(* CODESYS project INTERNA2 DRIVE TEST V17.project

Project tree, tasks and I/O mapping:
  Device : TX510-P3CV01, Turck, order no. 6828105, version 1.0.4.0
    application Application
      libraries: Standard, * (System); VisuDialogs, * (System); CAA File, * (CAA Technical Workgroup); CAA Real Time Clock Extern, * (CAA Technical Workgroup); SysTime23, 3.5.2.0 (System); NETWORK, 1.2.1.0 (OSCAT); SysTimeCore, * (System)
      task VISU_TASK (cyclic, interval 100 ms, priority 31) calls VisuElems.Visu_Prg
      task ENIPScannerServiceTask (cyclic, interval t#20ms, priority 30) calls EtherNet_IP_Scanner.ServiceCycle
      task MainTask (cyclic, interval t#20ms, priority 1) calls PLC_PRG
      task ENIPScannerIOTask (cyclic, interval t#10ms, priority 1) calls EtherNet_IP_Scanner.IOCycle
      task AlarmManagerTask (cyclic, interval 50 ms, priority 31) calls AlarmManager.Alarm_Prg
      visualisation PRINCIPAL
      visualisation Analog_Test
      visualisation Drive_Test
      program PLC_PRG [LD]
      global variables GLOBAL_VARS
      visualisation Test_DAQ
      program CSVMON_FILE_GEN [LD]
      Alarm Configuration
        alarm class Error (priority 10, acknowledge ACK)
        alarm class Warning (priority 30, acknowledge REP)
        alarm class Info (priority 100, acknowledge REP)
        AlarmStorage
        text list AlarmGroup
        alarm group AlarmGroup
            11 [Info]: Comparison Equal, ExpressionToCompare TRUE, Expression OPERACION.ROTADORES_INFO_MSG - "PARA ACCIONAR ROTADORES, MUEVA EL BUGGY HACIA EL SUR"
            8 [Info]: Comparison Equal, ExpressionToCompare TRUE, Expression PLC_PRG.ANY_ALARM - "PRESIONE EL BOTON CONFIRMAR PARA RESTABLECER"
            9 [Error]: Comparison Equal, ExpressionToCompare TRUE, Expression PLC_PRG.POWERFLEX_FAULT_ACTIVE - "FALLA DRIVE MOTOR BUGGY "
            19 [Info]: Comparison Equal, ExpressionToCompare TRUE, Expression PLC_PRG.HMI_AUTO_MODE - "INFO MODO AUTO: BUGGY DIRECCION NORTE, VELOCIDAD LENTA"
            10 [Error]: Comparison Equal, ExpressionToCompare TRUE, Expression PLC_PRG.REMOTE_MODULE2_FAULT - "L1: ERROR COMUNICACION MODULO GABINETE VARIADOR & FUERZA"
            15 [Warning]: Comparison Equal, ExpressionToCompare FALSE, Expression OPERACION.SW_ANTORCHA_EJEB - "LIMITE CABEZAL ANTORCHA EJEB ALCANZADO"
            18 [Error]: Comparison Equal, ExpressionToCompare TRUE, Expression PLC_PRG.WELDING_TRAVEL_FEEDBACK_FAULT - "ERROR EN GENERACION DE ARCO"
            16 [Warning]: Comparison Equal, ExpressionToCompare FALSE, Expression OPERACION.SW_BOOM_UP - "LIMITE BOOM SUPERIOR ALCANZADO"
            17 [Warning]: Comparison Equal, ExpressionToCompare FALSE, Expression OPERACION.SW_BOOM_DOWN - "LIMITE BOOM INFERIOR ALCANZADO"
            3 [Error]: Comparison Equal, ExpressionToCompare TRUE, Expression PLC_PRG.ENCODER_FAULT - "ERROR DE SINCRONIZACION BUGGY:REVISAR ENCODER"
            4 [Warning]: Comparison Equal, ExpressionToCompare FALSE, Expression PLC_PRG.SW_NORTE - "BUGGY LIMTE DE CARRERA NORTE ALCANZADO"
            5 [Warning]: Comparison Equal, ExpressionToCompare FALSE, Expression PLC_PRG.SW_SUR - "BUGGY LIMITE DE CARRERA SUR ALCANZADO"
            6 [Error]: Comparison Equal, ExpressionToCompare TRUE, Expression PLC_PRG.REMOTE_MODULE1_FAULT - "L0: ERROR COMUNICACION MODULO DETRAS HMI PRINCIPAL"
            7 [Warning]: Comparison Equal, ExpressionToCompare TRUE, Expression PLC_PRG.EMERGENCY_STOP_ACTIVE - "PARO DE EMERGENCIA EXTERNO ACTIVO"
            14 [Warning]: Comparison Equal, ExpressionToCompare FALSE, Expression OPERACION.SW_ANTORCHA_EJEA - "LIMITE CABEZAL ANTORCHA EJEA ALCANZADO"
            13 [Warning]: Comparison Equal, ExpressionToCompare FALSE, Expression OPERACION.SW_ANTORCHA_DOWN - "LIMITE CABEZAL ANTORCHA INFERIOR ALCANZADO"
            12 [Warning]: Comparison Equal, ExpressionToCompare FALSE, Expression OPERACION.SW_ANORTCHA_UP - "LIMITE CABEZAL ANTORCHA SUPERIOR ALCANZADO"
            20 [Error]: Comparison Equal, ExpressionToCompare TRUE, Expression PLC_PRG.REMOTE_MODULE3_FAULT - "L2: ERROR COMUNICACION MODULO GABINETE AUXILIAR,ANTORCHAS"
      program OPERACION [LD]
      visualisation OPERACION
      visualisation BUGGY
    Ethernet : Ethernet, Turck, version 3.5.7.20
        settings: IPAddress = [192,168,5,211]; SubnetMask = [255,255,255,0]; GatewayAddress = [0,0,0,0]; MACAddress = [16#00,16#00,16#00,16#00,16#00,16#00]; SaveCommunicationSettings = FALSE
      EtherNet_IP_Scanner : EtherNet/IP Scanner, 3S - Smart Software Solutions GmbH, order no. 1, version 3.5.7.0
          settings: IPAddress = [16#C0,16#A8,16#05,16#65]; SubnetMask = [16#00,16#00,16#00,16#00]; GatewayAddress = [16#00,16#00,16#00,16#00]; TCPFlags = 1; Options.Auto-Reestablish Connections = True
        REMOTE_MODULE1 : BL20-E-GW-EN, TURCK, order no. 6827329, version Major Revision=16#2, Minor Revision = 16#7
            settings: INITIALIZED = TRUE; IP address of Target = [16#C0,16#A8,16#05,16#67]; Keying.Compatibility Bit = TRUE; RequiredConfigVersion = 50660864; Number of Connections = 1; Connection Settings.Requested packet intervall (µs) = 10000; Connection Settings.OT Connection Parameters = 18442; Connection Settings.TO Connection Parameters = 10246; Connection Settings.Connection Flags = 1056; Connection Settings.Connection Path Size = 8; Connection Settings.Config#2 Size = 16; Configuration Data = [16#0,16#0,16#0,16#0,16#0,16#0,16#0,16#0,16#0,16#0,16#0,16#0,16#0,16#0,16#0,16#0]; Connection Path = [16#20,16#04,16#24,16#6A,16#2C,16#66,16#2C,16#65]; DI1_0_RESERVED.ReadOnly = False; DI1_0_RESERVED.BitSize = 16; DI1_0_RESERVED.DataSize = 2; DI1_1.ReadOnly = False; DI1_1.BitSize = 16; DI1_1.DataSize = 2; DO1_0_RESERVED.ReadOnly = False; DO1_0_RESERVED.BitSize = 16; DO1_0_RESERVED.DataSize = 2; D01_1.ReadOnly = False; D01_1.BitSize = 16; D01_1.DataSize = 2; DI1_0_RESERVED.Name = 'DI1_0_RESERVED'; DI1_0_RESERVED.HelpString = ''; DI1_0_RESERVED.ReadOnly = False; DI1_0_RESERVED.BitSize = 16; DI1_0_RESERVED.DataSize = 2; DI1_0_RESERVED.DataType = 'UINT'; DI1_1.Name = 'DI1_1'; DI1_1.HelpString = ''; DI1_1.ReadOnly = False; DI1_1.BitSize = 16; DI1_1.DataSize = 2; DI1_1.DataType = 'UINT'; DO1_0_RESERVED.Name = 'DO1_0_RESERVED'; DO1_0_RESERVED.HelpString = ''; DO1_0_RESERVED.ReadOnly = False;
              DO1_0_RESERVED.BitSize = 16; DO1_0_RESERVED.DataSize = 2; DO1_0_RESERVED.DataType = 'UINT'; D01_1.Name = 'D01_1'; D01_1.HelpString = ''; D01_1.ReadOnly = False; D01_1.BitSize = 16; D01_1.DataSize = 2; D01_1.DataType = 'UINT'; ConfigVersion = 50660864
            input  Application.PLC_PRG.EMERGENCY_STOP : BOOL  // DI1_1.Bit0
            input  Application.OPERACION.JOYUP : BOOL  // DI1_1.Bit1
            input  Application.OPERACION.JOYDOWN : BOOL  // DI1_1.Bit2
            input  Application.OPERACION.JOY_EJEA : BOOL  // DI1_1.Bit3
            input  Application.OPERACION.JOY_EJEB : BOOL  // DI1_1.Bit4
            input  Application.PLC_PRG.NA4_TRAVEL2 : BOOL  // DI1_1.Bit12
            input  Application.PLC_PRG.NA4_TRAVEL1 : BOOL  // DI1_1.Bit13
            input  Application.PLC_PRG.NA5_TRAVEL : BOOL  // DI1_1.Bit14
            input  Application.PLC_PRG.HEARTBEAT_RETURN : BOOL  // DI1_1.Bit15
            output Application.PLC_PRG.NA5_START : BOOL  // D01_1.Bit0
            output Application.PLC_PRG.NA4_START1 : BOOL  // D01_1.Bit1
            output Application.PLC_PRG.NA4_START2 : BOOL  // D01_1.Bit2
            output Application.PLC_PRG.NA_NOT_STOP : BOOL  // D01_1.Bit3
            output Application.PLC_PRG.HEARTBEAT_SEND : BOOL  // D01_1.Bit15
            unmapped channels: DI1_0_RESERVED, DI1_1, DO1_0_RESERVED, D01_1
        BUGGY_DRIVE : PowerFlex 525, Rockwell Automation - Allen-Bradley, order no. 25B..., version Major Revision=16#4, Minor Revision = 16#1
            settings: INITIALIZED = TRUE; IP address of Target = [16#C0,16#A8,16#05,16#66]; Keying.Check Vendor Code = FALSE; Keying.Check Product Code = FALSE; RequiredConfigVersion = 50660864; Number of Connections = 1; Connection Settings.Requested packet intervall (µs) = 10000; Connection Settings.OT Connection Parameters = 18442; Connection Settings.TO Connection Parameters = 18442; Connection Settings.Connection Flags = 1056; Connection Settings.Connection Path Size = 8; Connection Path = [16#20,16#04,16#24,16#06,16#2C,16#02,16#2C,16#01]; Reserved.ReadOnly = False; Reserved.BitSize = 32; Reserved.DataSize = 4; Logic Status 0.ReadOnly = False; Logic Status 0.BitSize = 16; Logic Status 0.DataSize = 2; Feedback 0.ReadOnly = False; Feedback 0.BitSize = 16; Feedback 0.DataSize = 2; Logic Command 0.ReadOnly = False; Logic Command 0.BitSize = 16; Logic Command 0.DataSize = 2; Reference 0.ReadOnly = False; Reference 0.BitSize = 16; Reference 0.DataSize = 2; Reserved.Name = 'Reserved'; Reserved.HelpString = ''; Reserved.ReadOnly = False; Reserved.BitSize = 32; Reserved.DataSize = 4; Reserved.DataType = 'DWORD'; Logic Status 0.Name = 'Logic Status 0'; Logic Status 0.HelpString = 'Drive 0 Logic Status'; Logic Status 0.ReadOnly = False; Logic Status 0.BitSize = 16; Logic Status 0.DataSize = 2; Logic Status 0.DataType = 'WORD'; Feedback 0.Name = 'Feedback 0';
              Feedback 0.HelpString = 'Drive 0 Feedback'; Feedback 0.ReadOnly = False; Feedback 0.BitSize = 16; Feedback 0.DataSize = 2; Feedback 0.DataType = 'WORD'; Logic Command 0.Name = 'Logic Command 0'; Logic Command 0.HelpString = 'Drive 0 Logic Command'; Logic Command 0.ReadOnly = False; Logic Command 0.BitSize = 16; Logic Command 0.DataSize = 2; Logic Command 0.DataType = 'WORD'; Reference 0.Name = 'Reference 0'; Reference 0.HelpString = 'Drive 0 Reference'; Reference 0.ReadOnly = False; Reference 0.BitSize = 16; Reference 0.DataSize = 2; Reference 0.DataType = 'WORD'; ConfigVersion = 50660864
            input  Application.PLC_PRG.PWRFLEX_LOGIC_STATUS : WORD  // Logic Status 0
            input  Application.PLC_PRG.PWRFLEX_FEEDBACK : WORD  // Feedback 0
            output Application.PLC_PRG.PWRFLEX_LOGIC_CMD : WORD  // Logic Command 0
            output Application.PLC_PRG.PWRFLEX_SPEEDREF : WORD  // Reference 0
            unmapped channels: Reserved
        In_Sight_Micro_1000_Series : In-Sight Micro 1000 Series, Cognex, order no. ism1XXX, version Major Revision=16#a, Minor Revision = 16#1
            settings: INITIALIZED = TRUE; IP address of Target = [16#C0,16#A8,16#05,16#04]; Keying.Compatibility Bit = TRUE; RequiredConfigVersion = 50660864; Number of Connections = 1; Connection Settings.Requested packet intervall (µs) = 10000; Connection Settings.OT Connection Parameters = 18434; Connection Settings.TO Connection Parameters = 10258; Connection Settings.Connection Flags = 1062; Connection Settings.Connection Path Size = 8; Connection Path = [16#20,16#04,16#24,16#01,16#2C,16#FE,16#2C,16#0C]; Generic Parameter1.ReadOnly = False; Generic Parameter1.BitSize = 32; Generic Parameter1.DataSize = 4; Generic Parameter3.ReadOnly = False; Generic Parameter3.BitSize = 32; Generic Parameter3.DataSize = 4; Generic Parameter2.ReadOnly = False; Generic Parameter2.BitSize = 32; Generic Parameter2.DataSize = 4; Generic Parameter4.ReadOnly = False; Generic Parameter4.BitSize = 32; Generic Parameter4.DataSize = 4; Generic Parameter1.Name = 'Generic Parameter1'; Generic Parameter1.HelpString = ''; Generic Parameter1.ReadOnly = False; Generic Parameter1.BitSize = 32; Generic Parameter1.DataSize = 4; Generic Parameter1.DataType = 'REAL'; Generic Parameter3.Name = 'Generic Parameter3'; Generic Parameter3.HelpString = ''; Generic Parameter3.ReadOnly = False; Generic Parameter3.BitSize = 32; Generic Parameter3.DataSize = 4; Generic Parameter3.DataType = 'REAL'; Generic Parameter2.Name = 'Generic Parameter2'; Generic Parameter2.HelpString = ''; Generic Parameter2.ReadOnly = False; Generic Parameter2.BitSize = 32; Generic Parameter2.DataSize = 4;
              Generic Parameter2.DataType = 'REAL'; Generic Parameter4.Name = 'Generic Parameter4'; Generic Parameter4.HelpString = ''; Generic Parameter4.ReadOnly = False; Generic Parameter4.BitSize = 32; Generic Parameter4.DataSize = 4; Generic Parameter4.DataType = 'REAL'; ConfigVersion = 50660864
            input  Application.PLC_PRG.COGNEX_AUX1 : REAL  // Generic Parameter1
            input  Application.PLC_PRG.COGNEX_AUX2 : REAL  // Generic Parameter3
            input  Application.PLC_PRG.COGNEX_AUX3 : REAL  // Generic Parameter2
            input  Application.PLC_PRG.COGNEX_AUX4 : REAL  // Generic Parameter4
        REMOTE_MODULE2 : BL20-E-GW-EN, TURCK, order no. 6827329, version Major Revision=16#2, Minor Revision = 16#7
            settings: INITIALIZED = TRUE; IP address of Target = [16#C0,16#A8,16#05,16#69]; Keying.Compatibility Bit = TRUE; RequiredConfigVersion = 50660864; Number of Connections = 1; Connection Settings.Requested packet intervall (µs) = 10000; Connection Settings.OT Connection Parameters = 18442; Connection Settings.TO Connection Parameters = 10246; Connection Settings.Connection Flags = 1056; Connection Settings.Connection Path Size = 8; Connection Settings.Config#2 Size = 16; Configuration Data = [16#0,16#0,16#0,16#0,16#0,16#0,16#0,16#0,16#0,16#0,16#0,16#0,16#0,16#0,16#0,16#0]; Connection Path = [16#20,16#04,16#24,16#6A,16#2C,16#66,16#2C,16#65]; DI2_0_RESERVED.ReadOnly = False; DI2_0_RESERVED.BitSize = 16; DI2_0_RESERVED.DataSize = 2; DI2_1.ReadOnly = False; DI2_1.BitSize = 16; DI2_1.DataSize = 2; DO2_0_RESERVED.ReadOnly = False; DO2_0_RESERVED.BitSize = 16; DO2_0_RESERVED.DataSize = 2; DO2_1.ReadOnly = False; DO2_1.BitSize = 16; DO2_1.DataSize = 2; DI2_0_RESERVED.Name = 'DI2_0_RESERVED'; DI2_0_RESERVED.HelpString = ''; DI2_0_RESERVED.ReadOnly = False; DI2_0_RESERVED.BitSize = 16; DI2_0_RESERVED.DataSize = 2; DI2_0_RESERVED.DataType = 'UINT'; DI2_1.Name = 'DI2_1'; DI2_1.HelpString = ''; DI2_1.ReadOnly = False; DI2_1.BitSize = 16; DI2_1.DataSize = 2; DI2_1.DataType = 'UINT'; DO2_0_RESERVED.Name = 'DO2_0_RESERVED'; DO2_0_RESERVED.HelpString = ''; DO2_0_RESERVED.ReadOnly = False;
              DO2_0_RESERVED.BitSize = 16; DO2_0_RESERVED.DataSize = 2; DO2_0_RESERVED.DataType = 'UINT'; DO2_1.Name = 'DO2_1'; DO2_1.HelpString = ''; DO2_1.ReadOnly = False; DO2_1.BitSize = 16; DO2_1.DataSize = 2; DO2_1.DataType = 'UINT'; ConfigVersion = 50660864
            input  Application.OPERACION.SW_BOOM_DOWN : BOOL  // DI2_1.Bit0
            input  Application.OPERACION.SW_BOOM_UP : BOOL  // DI2_1.Bit1
            input  Application.PLC_PRG.HEARTBEAT_RETURN2 : BOOL  // DI2_1.Bit15
            output Application.OPERACION.CONVEYOR_NORTE_L02_KM1 : BOOL  // DO2_1.Bit0
            output Application.OPERACION.CONVEYOR_SUR_L02_KM2 : BOOL  // DO2_1.Bit1
            output Application.OPERACION.ROTADORES_EJEA_L02_KM3 : BOOL  // DO2_1.Bit2
            output Application.OPERACION.ROTADORES_EJEB_L02_KM4 : BOOL  // DO2_1.Bit3
            output Application.OPERACION.BOOM_DOWN_KM6 : BOOL  // DO2_1.Bit4
            output Application.OPERACION.BOOM_UP_KM5 : BOOL  // DO2_1.Bit5
            output Application.OPERACION.ASPIRADORA_KM7 : BOOL  // DO2_1.Bit6
            output Application.OPERACION.RELAY_BRAZO_TIERRAS_UP : BOOL  // DO2_1.Bit7
            output Application.OPERACION.RELAY_BRAZO_TIERRAS_DOWN : BOOL  // DO2_1.Bit8
            output Application.PLC_PRG.HEARTBEAT_SEND2 : BOOL  // DO2_1.Bit15
            unmapped channels: DI2_0_RESERVED, DI2_1, DO2_0_RESERVED, DO2_1
        REMOTE_MODULE3 : BL20-E-GW-EN, TURCK, order no. 6827329, version Major Revision=16#2, Minor Revision = 16#7
            settings: INITIALIZED = TRUE; IP address of Target = [16#C0,16#A8,16#05,16#6A]; Keying.Compatibility Bit = TRUE; RequiredConfigVersion = 50660864; Number of Connections = 1; Connection Settings.Requested packet intervall (µs) = 10000; Connection Settings.OT Connection Parameters = 18442; Connection Settings.TO Connection Parameters = 18438; Connection Settings.Connection Flags = 1056; Connection Settings.Connection Path Size = 8; Connection Settings.Config#2 Size = 16; Configuration Data = [16#0,16#0,16#0,16#0,16#0,16#0,16#0,16#0,16#0,16#0,16#0,16#0,16#0,16#0,16#0,16#0]; Connection Path = [16#20,16#04,16#24,16#6A,16#2C,16#66,16#2C,16#65]; DI3_0_RESERVED.ReadOnly = False; DI3_0_RESERVED.BitSize = 16; DI3_0_RESERVED.DataSize = 2; DI3_1.ReadOnly = False; DI3_1.BitSize = 16; DI3_1.DataSize = 2; DO3_0_RESERVED.ReadOnly = False; DO3_0_RESERVED.BitSize = 16; DO3_0_RESERVED.DataSize = 2; DO3_1.ReadOnly = False; DO3_1.BitSize = 16; DO3_1.DataSize = 2; DI3_0_RESERVED.Name = 'DI3_0_RESERVED'; DI3_0_RESERVED.HelpString = ''; DI3_0_RESERVED.ReadOnly = False; DI3_0_RESERVED.BitSize = 16; DI3_0_RESERVED.DataSize = 2; DI3_0_RESERVED.DataType = 'UINT'; DI3_1.Name = 'DI3_1'; DI3_1.HelpString = ''; DI3_1.ReadOnly = False; DI3_1.BitSize = 16; DI3_1.DataSize = 2; DI3_1.DataType = 'UINT'; DO3_0_RESERVED.Name = 'DO3_0_RESERVED'; DO3_0_RESERVED.HelpString = ''; DO3_0_RESERVED.ReadOnly = False;
              DO3_0_RESERVED.BitSize = 16; DO3_0_RESERVED.DataSize = 2; DO3_0_RESERVED.DataType = 'UINT'; DO3_1.Name = 'DO3_1'; DO3_1.HelpString = ''; DO3_1.ReadOnly = False; DO3_1.BitSize = 16; DO3_1.DataSize = 2; DO3_1.DataType = 'UINT'; ConfigVersion = 50660864
            input  Application.PLC_PRG.SW_NORTE : BOOL  // DI3_1.Bit0
            input  Application.PLC_PRG.SW_SUR : BOOL  // DI3_1.Bit1
            input  Application.OPERACION.SW_ANORTCHA_UP : BOOL  // DI3_1.Bit2
            input  Application.OPERACION.SW_ANTORCHA_DOWN : BOOL  // DI3_1.Bit3
            input  Application.OPERACION.SW_ANTORCHA_EJEA : BOOL  // DI3_1.Bit4
            input  Application.OPERACION.SW_ANTORCHA_EJEB : BOOL  // DI3_1.Bit5
            input  Application.PLC_PRG.HEARTBEAT_RETURN3 : BOOL  // DI3_1.Bit15
            output Application.OPERACION.RELAY_VALVULA1 : BOOL  // DO3_1.Bit0
            output Application.OPERACION.RELAY_VALVULA2 : BOOL  // DO3_1.Bit1
            output Application.OPERACION.TOLVA_ON : BOOL  // DO3_1.Bit4
            output Application.OPERACION.CAMARA_ON : BOOL  // DO3_1.Bit5
            output Application.OPERACION.ANTORCHA_EJEA : BOOL  // DO3_1.Bit6
            output Application.OPERACION.ANTORCHA_EJEB : BOOL  // DO3_1.Bit7
            output Application.OPERACION.ANTORCHA_UP : BOOL  // DO3_1.Bit8
            output Application.OPERACION.ANTORCHA_DOWN : BOOL  // DO3_1.Bit9
            output Application.PLC_PRG.HEARTBEAT_SEND3 : BOOL  // DO3_1.Bit15
            unmapped channels: DI3_0_RESERVED, DI3_1, DO3_0_RESERVED, DO3_1
  libraries: VisuSymbols, 3.5.10.0 (System)
  text list GlobalTextList
  text list System
*)

// Device/Application/GLOBAL_VARS
{attribute 'qualified_only'}
VAR_GLOBAL
	  uiFileStdState:     UINT;  //TEXT CMD STATE
	  sFileName: 		  STRING;		//FILE NAM STRING (DIRECTORY+DATA)
	  sFileWriteString:	  STRING;
	
	  
END_VAR

// Device/Application/PLC_PRG
PROGRAM PLC_PRG
VAR
(* 
======>instalar librerias:
1)network(OSCAT 1.2.1.0)
2)CAA FILE 3.5.7.0
3) SYSTIME32 3.5.2.0
*)	

//--BL20 VARS--

//EL SIGUIENTE DIRECCIONAMIENTO NO ES RECOMENDADO, LA DIRECCION PUEDE SER REASIGNADA 
//AL AGREGAR UN DISPOSITIVO:
//	IN00 AT %IB102 :BYTE;
//	IN01 AT %IB103 :BYTE;
//-----DIGITAL-----
//INPUTS
DI1_1 :USINT;
//OUTPUTS
DO1_1 :USINT;

//----ANALOG------
//INPUTS
ANA_INPUT1_1 :INT;
ANA_INPUT1_2 :INT;
//OUTPUTS

//VARS
ANA_IN_AUX1 :REAL;
ANA_AMPS :REAL;

ANA_IN_AUX2 :REAL;


//-----------------------------------POWERFLEX VARS-----------------------------------------//
//MISCELLANEUS
PWRFLEX_START_CMD  :UINT; //16bit integer
PWRFLEX_STOP_CMD  :UINT; 
PWRFLEX_SPEEDREF_AUX :REAL;
PWRFLEX_SPEEDREF_AUX2 :REAL;
PWRFLEX_FEEDBACK :UINT;
PWRFLEX_FEEDBACK_AUX :REAL;
PWRFLEX_FEEDBACK_AUX2 :REAL;
PWRFLEX_FEEDBACK_AUX_OFFSET :REAL;

PWRFLEX_FEEDBACK_AUX3 :REAL;
PWRFLEX_FEEDBACK_AUX4 :REAL;

PWRFLEX_AMPS :REAL;
PWRFLEX_giro :BOOL;

PWRFLEX_AMPS_AUX :REAL;

//START =>26
//STOP =>9

//INPUTS
PWRFLEX_LOGIC_STATUS :WORD;

//OUTPUTS
PWRFLEX_LOGIC_CMD :WORD;
PWRFLEX_OPERATOR_START: BOOL;
PWRFLEX_OPERATOR_STOP: BOOL;
HMI_PWRFLEX_OPERATOR_STOP: BOOL;
PWRFLEX_START_STOP :BOOL;
PWRFLEX_SPEEDREF :WORD;

//----------------------------PROGRAM GENERAL MISCELLANEUS VARS------------------------------//
//->SQUARE GEN - PERIOD:1SEG
TIMER1_A: TON;
TIMER1_B: TON;


ALWAYS_OFF :BOOL:=FALSE;
VAR1 :BOOL;
VAR2 :BOOL;
VAR3 :BOOL;
//declare and assign value example
 //VARx :BOOL :=TRUE;

//----------------------------COGNEX VARS------------------------------//
In_Sight_Micro_1000_Series :DWORD;
COGNEX_AUX :DWORD;
COGNEX_AUX1 :REAL;
COGNEX_AUX2 :REAL;
COGNEX_AUX3 :REAL;
COGNEX_AUX4 :REAL;



//----------------------------TEXT VARS------------------------------//
TXT_CMD_ENABLE: BOOL;
TXT_CMD_SELECT: USINT;


TEST_TEXT: STRING;

TEXT: STRING;
TEST_BIT: BOOL;
TEST_BIT2: BOOL;



TON1: TON;
SAMPLING_TRIGGER: BOOL;


//----------------------------ALARMS------------------------------//
(*
ALARM_ERROR1: BOOL;
ALARM_WARNING1: BOOL;
ALARM_INFO1: BOOL;
*)
ACK_ALARM: BOOL;
ANY_ALARM: BOOL:=FALSE;
(*
ALARM_ERROR1_ACTIVE: BOOL;
ALARM_WARNING1_ACTIVE: BOOL;
ALARM_INFO1_ACTIVE: BOOL;
*)
//-----EMERGENCY STOP----
EMERGENCY_STOP: BOOL;
EMERGENCY_STOP_ACTIVE: BOOL;
HMI_EMERGENCY_STOP: BOOL;
HMI_EMERGENCY_STOP_ACTIVE: BOOL;

//----DRIVE FAULT-------
POWERFLEX_FAULT_ACTIVE: BOOL;

//------ENCODER---------
ENCODER_FAULT_TON: TON;
ENCODER_FAULT: BOOL;
ENCODER_FAULT_AUX: BOOL;
PWRFLEX_SPEED_DEVIATION: REAL;

//------LIMIT SWITCH BUGGY
SW_NORTE: BOOL;
SW_NORTE_FAULT: BOOL;
SW_NORTE_FALLING_TRIGGER: F_TRIG;
SW_SUR: BOOL;
SW_SUR_FAULT: BOOL;
SW_SUR_FALLING_TRIGGER: F_TRIG;

BUGGY_NORTE_ENABLE: BOOL;
BUGGY_NORTE_DISABLE: BOOL;
BUGGY_SUR_ENABLE: BOOL;
BUGGY_SUR_DISABLE: BOOL;
BUGGY_SUR_NORTE_ENABLE: BOOL;
BUGGY_SUR_NORTE_DISABLE: BOOL;

//----------REMOTE MODULE COMMUNICATION ERROR------------
//>>MODULE1 (L0)

HEARTBEAT_SEND: BOOL;
HEARTBEAT_RETURN: BOOL;
REMOTE_MODULE1_FAULT: BOOL;
REMOTE_MODULE1_FAULT_AUX: BOOL;

TIMER_HEARTBEAT_FEEDBACK1: TON;
TIMER_HEARTBEAT_FEEDBACK2: TON;

//-----MODULE 2 COMUNICATION ERROR (L1)
HEARTBEAT_SEND2: BOOL;
HEARTBEAT_RETURN2: BOOL;
REMOTE_MODULE2_FAULT: BOOL;
REMOTE_MODULE2_FAULT_AUX: BOOL;

TIMER_HEARTBEAT_FEEDBACK1_2: TON;
TIMER_HEARTBEAT_FEEDBACK2_2: TON;

//-----MODULE 3 COMUNICATION ERROR (L2)
HEARTBEAT_SEND3: BOOL;
HEARTBEAT_RETURN3: BOOL;
REMOTE_MODULE3_FAULT: BOOL;
REMOTE_MODULE3_FAULT_AUX: BOOL;

TIMER_HEARTBEAT_FEEDBACK1_3: TON;
TIMER_HEARTBEAT_FEEDBACK2_3: TON;

//-------WELDING SEQUENCE ERROR
WELDING_TRAVEL_FEEDBACK: TON;
WELDING_TRAVEL_FEEDBACK_FAULT: BOOL;



//-----------------------------
OPERATOR_CONFIRM_ERROR: BOOL;

//-----------------OPERATOR------------------

BUGGY_SPEED_SELECTOR: BOOL;
BUGGY_SPEED_FAST: REAL:=400.0;
BUGGY_SPEED_SLOW: REAL:=30.0;
BUGGY_SPEED: REAL;
BUGGY_SPEED_AUX1: REAL;
BUGGY_SPEED_FEEDBACK_OFFSET: REAL:=1.0;
BUGGY_SPEED_FEEDBACK_OFFSET_AUX: REAL;
BUGGY_SPEED_REFERENCE_OFFSET: REAL:=1.0;
BUGGY_SPEED_REFERENCE_OFFSET_AUX: REAL;

//------------NA CONTROL-------------
HMI_AUTO_MODE: BOOL;
NA_AUTO_MODE: BOOL;

//NA INPUTS
NA5_TRAVEL: BOOL;  //DC WELDING ACTIVE
NA4_TRAVEL1: BOOL; //AC1 WELDING ACTIVE
NA4_TRAVEL2: BOOL; //AC2 WELDING ACTIVE

//OUTPUTS TO NA
NA5_START: BOOL; //DC START
NA4_START1: BOOL; //AC1 START
NA4_START2: BOOL; //AC2 START

ACTIVATE_NA_WELDING_SEQUENCE: BOOL;
ACTIVATE_NA5_DC: TON; //START DELAY DC
ACTIVATE_NA4_AC1: TON; //START DELAY AC1
ACTIVATE_NA4_AC2: TON; //START DELAY AC1

ALL_NA_TRAVEL_OK: BOOL;

NA_NOT_STOP: BOOL; //PLC STOP TO ALL NA´S

//WELDING AUTO MODE
AUTO_MODE_PERMISSIVES_OK: BOOL;
ASPIRADORA_AUTO_ON: BOOL;

AUTO_MODE_ARC_SELECT: BOOL; //FALSE=2 ARCOS, TRUE=3 ARCOS
AUTO_MODE_BYPASS: BOOL; //BYPASS PARA ACTIVAR ARCOS EN MODO MANUAL

END_VAR
VAR // added by the converter: edge detectors and wires of the graphical bodies
    _w1, _w2, _w3, _w4 : BOOL;
END_VAR

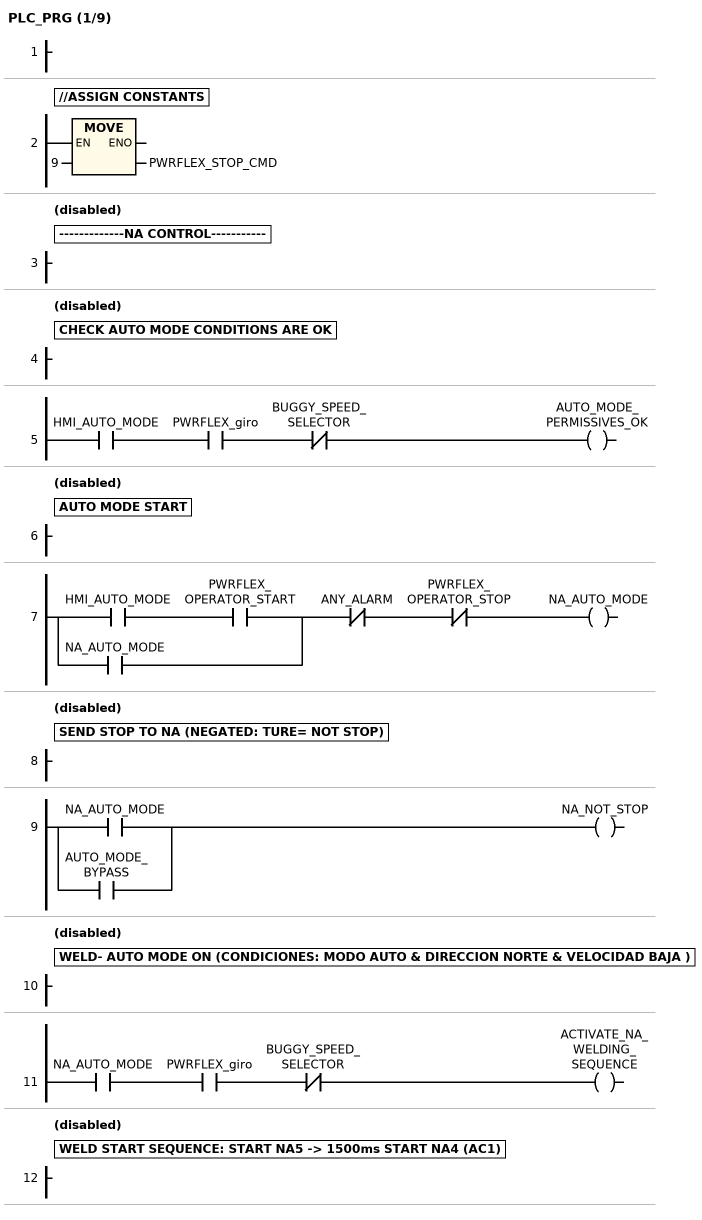
// NETWORK 1

// NETWORK 2
// label: //ASSIGN CONSTANTS
PWRFLEX_STOP_CMD := 9;

// NETWORK 3 (disabled)
// label: -------------NA CONTROL-----------

// NETWORK 4 (disabled)
// label: CHECK AUTO MODE CONDITIONS ARE OK

// NETWORK 5
AUTO_MODE_PERMISSIVES_OK := HMI_AUTO_MODE AND PWRFLEX_giro AND NOT BUGGY_SPEED_SELECTOR;

// NETWORK 6 (disabled)
// label: AUTO MODE START

// NETWORK 7
NA_AUTO_MODE := (HMI_AUTO_MODE AND PWRFLEX_OPERATOR_START OR NA_AUTO_MODE) AND NOT ANY_ALARM AND NOT PWRFLEX_OPERATOR_STOP;

// NETWORK 8 (disabled)
// label: SEND STOP TO NA (NEGATED: TURE= NOT STOP)

// NETWORK 9
NA_NOT_STOP := NA_AUTO_MODE OR AUTO_MODE_BYPASS;

// NETWORK 10 (disabled)
// label: WELD- AUTO MODE ON (CONDICIONES: MODO AUTO & DIRECCION NORTE & VELOCIDAD BAJA )

// NETWORK 11
ACTIVATE_NA_WELDING_SEQUENCE := NA_AUTO_MODE AND PWRFLEX_giro AND NOT BUGGY_SPEED_SELECTOR;

// NETWORK 12 (disabled)
// label: WELD START SEQUENCE: START NA5 -> 1500ms START NA4 (AC1)

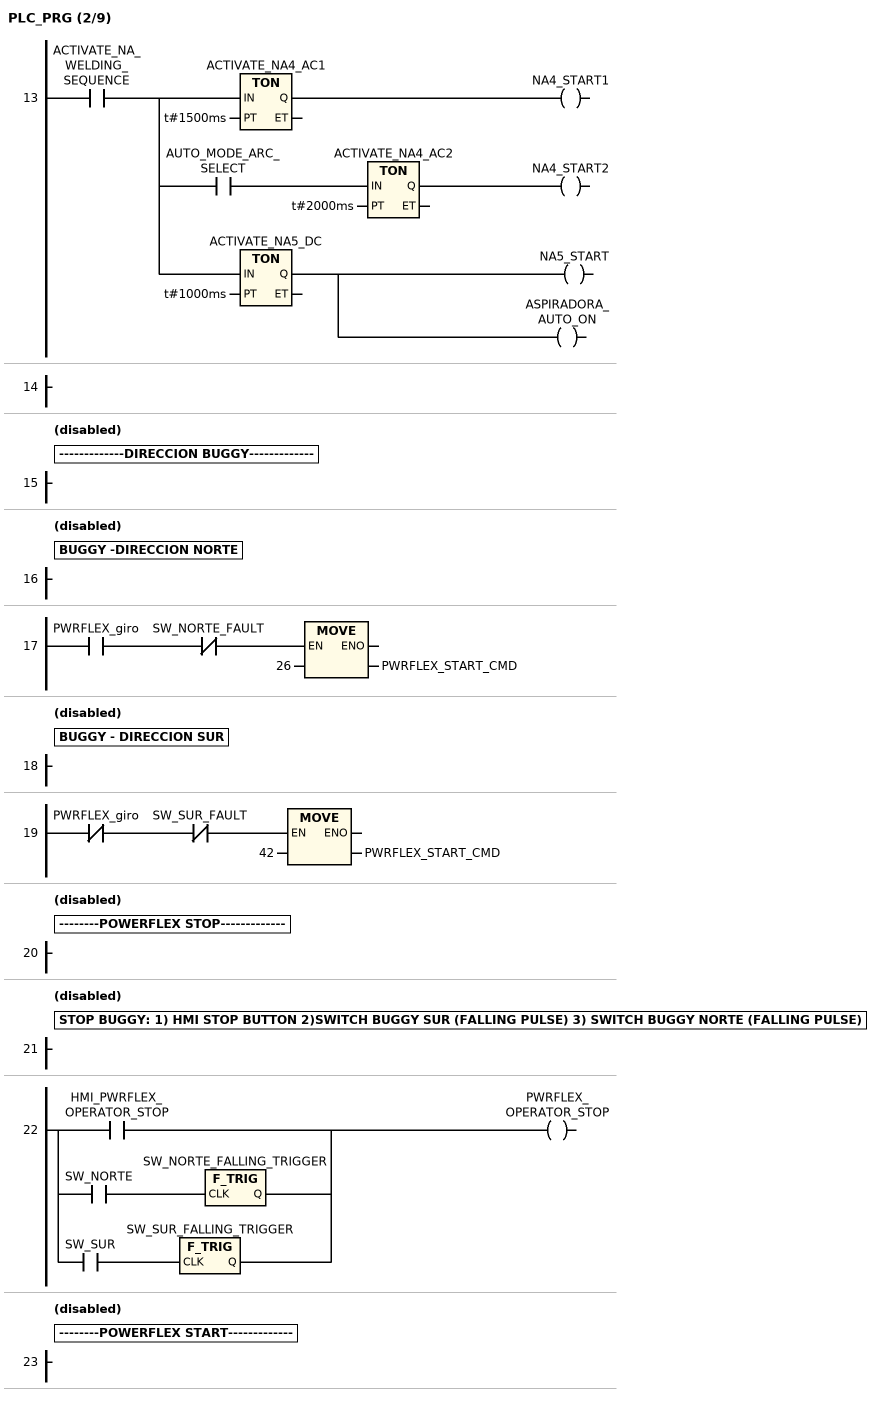
// NETWORK 13
ACTIVATE_NA4_AC1(IN := ACTIVATE_NA_WELDING_SEQUENCE, PT := t#1500ms); // TON
NA4_START1 := ACTIVATE_NA4_AC1.Q;
ACTIVATE_NA4_AC2(IN := ACTIVATE_NA_WELDING_SEQUENCE AND AUTO_MODE_ARC_SELECT, PT := t#2000ms); // TON
NA4_START2 := ACTIVATE_NA4_AC2.Q;
ACTIVATE_NA5_DC(IN := ACTIVATE_NA_WELDING_SEQUENCE, PT := t#1000ms); // TON
NA5_START := ACTIVATE_NA5_DC.Q;
ASPIRADORA_AUTO_ON := ACTIVATE_NA5_DC.Q;

// NETWORK 14

// NETWORK 15 (disabled)
// label: -------------DIRECCION BUGGY-------------

// NETWORK 16 (disabled)
// label: BUGGY -DIRECCION NORTE

// NETWORK 17
IF PWRFLEX_giro AND NOT SW_NORTE_FAULT THEN PWRFLEX_START_CMD := 26; END_IF

// NETWORK 18 (disabled)
// label: BUGGY - DIRECCION SUR

// NETWORK 19
IF NOT PWRFLEX_giro AND NOT SW_SUR_FAULT THEN PWRFLEX_START_CMD := 42; END_IF

// NETWORK 20 (disabled)
// label: --------POWERFLEX STOP-------------

// NETWORK 21 (disabled)
// label: STOP BUGGY: 1) HMI STOP BUTTON 2)SWITCH BUGGY SUR (FALLING PULSE) 3) SWITCH BUGGY NORTE (FALLING PULSE)

// NETWORK 22
SW_NORTE_FALLING_TRIGGER(CLK := SW_NORTE); // F_TRIG
SW_SUR_FALLING_TRIGGER(CLK := SW_SUR); // F_TRIG
PWRFLEX_OPERATOR_STOP := HMI_PWRFLEX_OPERATOR_STOP OR SW_NORTE_FALLING_TRIGGER.Q OR SW_SUR_FALLING_TRIGGER.Q;

// NETWORK 23 (disabled)
// label: --------POWERFLEX START-------------

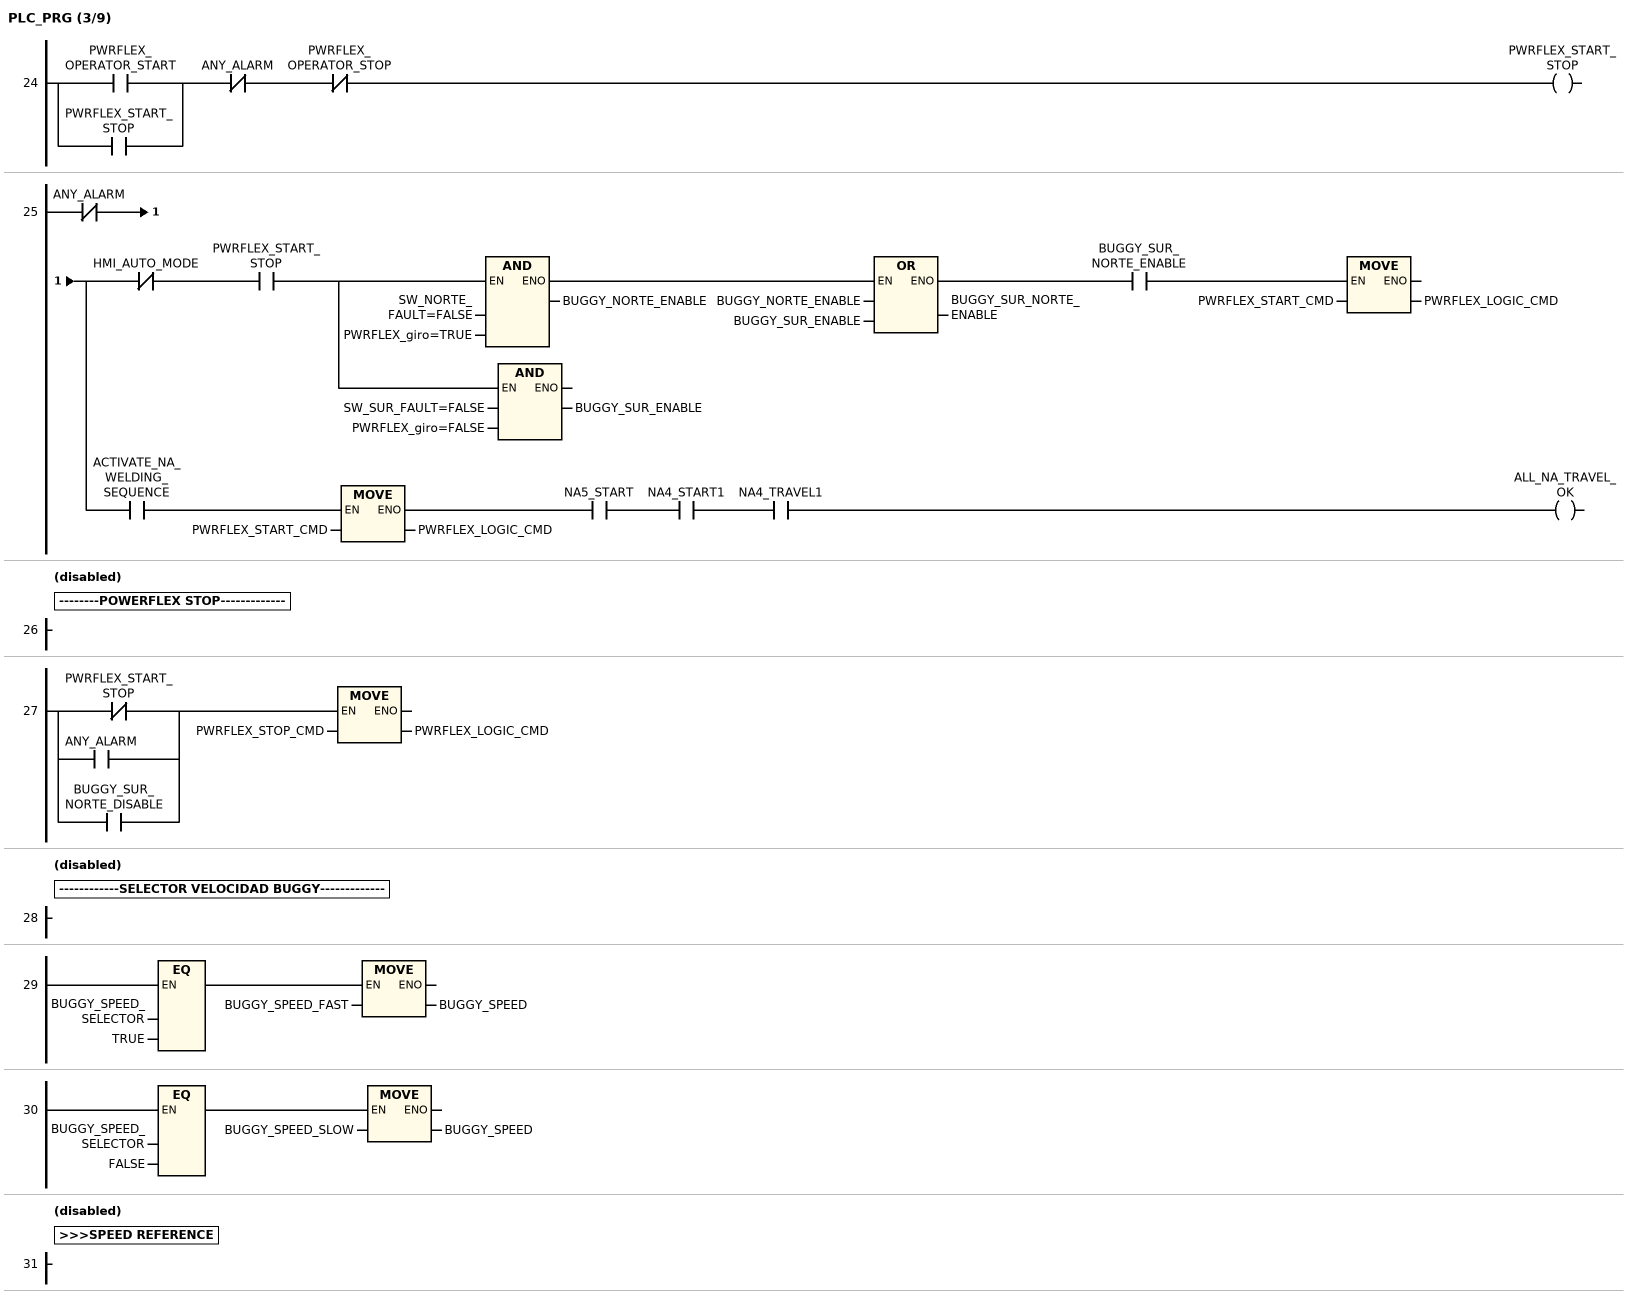
// NETWORK 24
PWRFLEX_START_STOP := (PWRFLEX_OPERATOR_START OR PWRFLEX_START_STOP) AND NOT ANY_ALARM AND NOT PWRFLEX_OPERATOR_STOP;

// NETWORK 25
_w1 := NOT ANY_ALARM;
_w2 := _w1 AND NOT HMI_AUTO_MODE AND PWRFLEX_START_STOP;
IF _w2 THEN BUGGY_NORTE_ENABLE := (SW_NORTE_FAULT=FALSE) AND (PWRFLEX_giro=TRUE); END_IF
IF _w2 THEN BUGGY_SUR_NORTE_ENABLE := BUGGY_NORTE_ENABLE OR BUGGY_SUR_ENABLE; END_IF
IF _w2 AND BUGGY_SUR_NORTE_ENABLE THEN PWRFLEX_LOGIC_CMD := PWRFLEX_START_CMD; END_IF
IF _w2 THEN BUGGY_SUR_ENABLE := (SW_SUR_FAULT=FALSE) AND (PWRFLEX_giro=FALSE); END_IF
IF _w1 AND ACTIVATE_NA_WELDING_SEQUENCE THEN PWRFLEX_LOGIC_CMD := PWRFLEX_START_CMD; END_IF
ALL_NA_TRAVEL_OK := (_w1 AND ACTIVATE_NA_WELDING_SEQUENCE) AND NA5_START AND NA4_START1 AND NA4_TRAVEL1;

// NETWORK 26 (disabled)
// label: --------POWERFLEX STOP-------------

// NETWORK 27
IF NOT PWRFLEX_START_STOP OR ANY_ALARM OR BUGGY_SUR_NORTE_DISABLE THEN
    PWRFLEX_LOGIC_CMD := PWRFLEX_STOP_CMD;
END_IF

// NETWORK 28 (disabled)
// label: ------------SELECTOR VELOCIDAD BUGGY-------------

// NETWORK 29
IF BUGGY_SPEED_SELECTOR = TRUE THEN BUGGY_SPEED := BUGGY_SPEED_FAST; END_IF

// NETWORK 30
IF BUGGY_SPEED_SELECTOR = FALSE THEN BUGGY_SPEED := BUGGY_SPEED_SLOW; END_IF

// NETWORK 31 (disabled)
// label: >>>SPEED REFERENCE

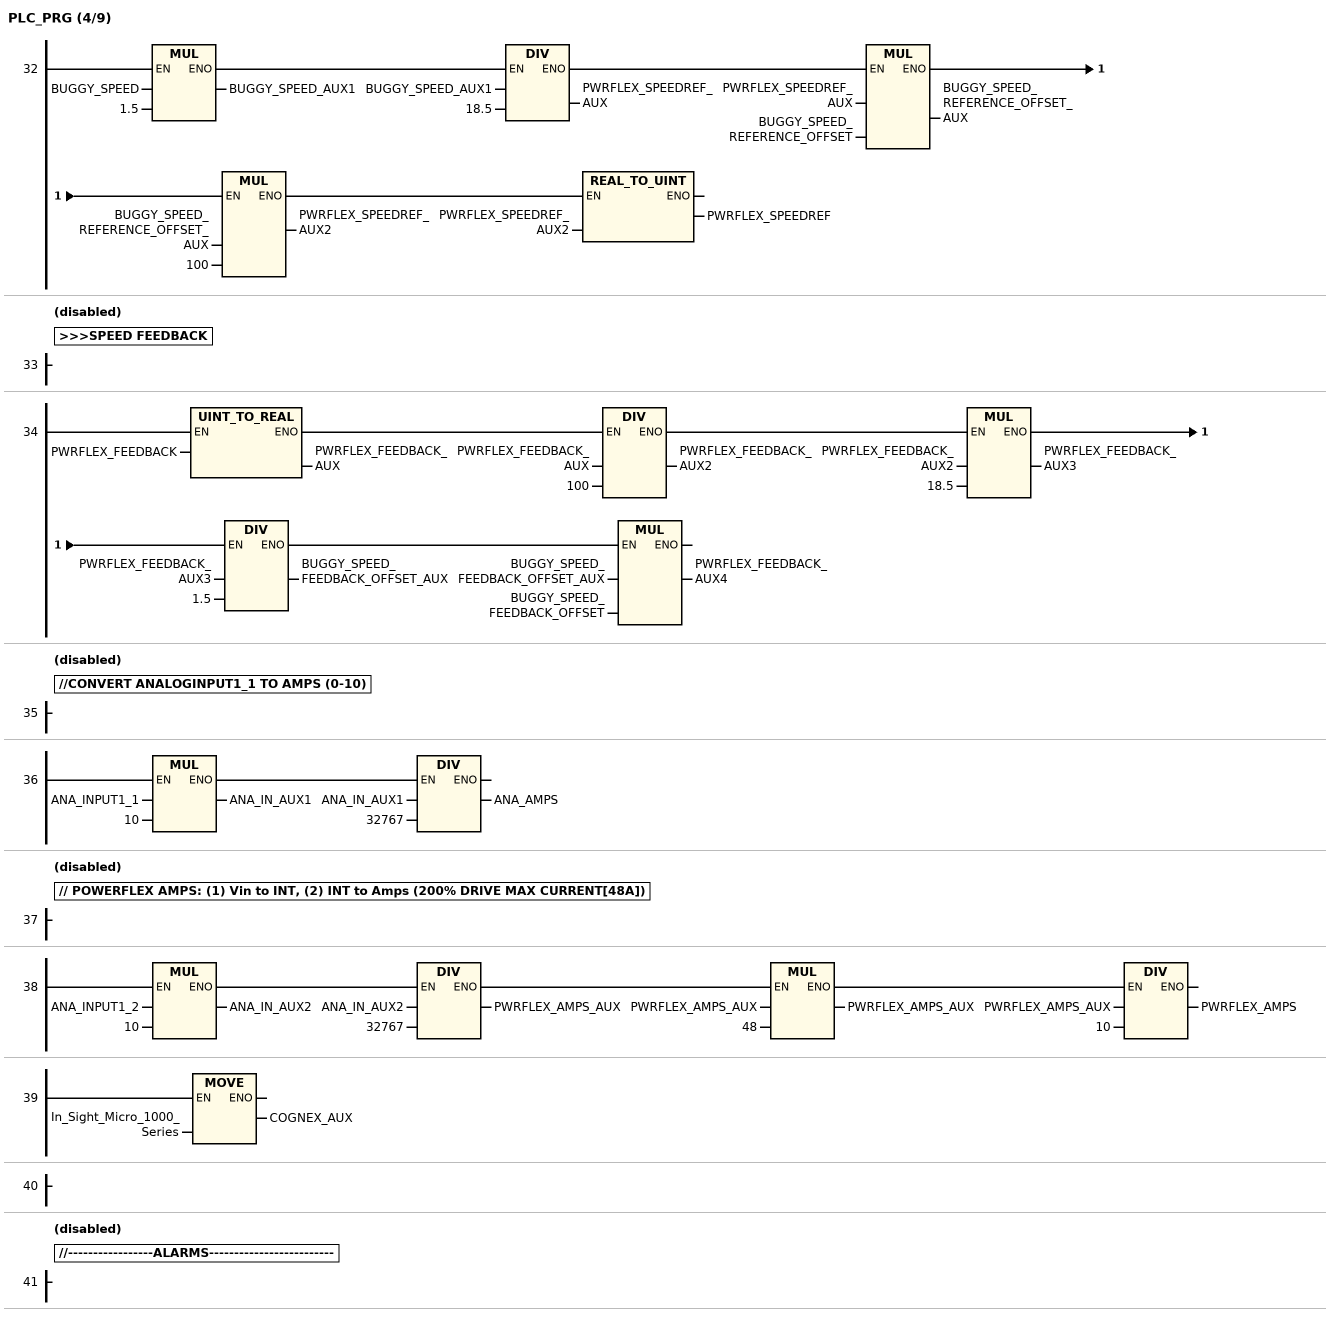
// NETWORK 32
BUGGY_SPEED_AUX1 := BUGGY_SPEED * 1.5;
PWRFLEX_SPEEDREF_AUX := BUGGY_SPEED_AUX1 / 18.5;
BUGGY_SPEED_REFERENCE_OFFSET_AUX := PWRFLEX_SPEEDREF_AUX * BUGGY_SPEED_REFERENCE_OFFSET;
PWRFLEX_SPEEDREF_AUX2 := BUGGY_SPEED_REFERENCE_OFFSET_AUX * 100;
PWRFLEX_SPEEDREF := REAL_TO_UINT(PWRFLEX_SPEEDREF_AUX2);

// NETWORK 33 (disabled)
// label: >>>SPEED FEEDBACK

// NETWORK 34
PWRFLEX_FEEDBACK_AUX := UINT_TO_REAL(PWRFLEX_FEEDBACK);
PWRFLEX_FEEDBACK_AUX2 := PWRFLEX_FEEDBACK_AUX / 100;
PWRFLEX_FEEDBACK_AUX3 := PWRFLEX_FEEDBACK_AUX2 * 18.5;
BUGGY_SPEED_FEEDBACK_OFFSET_AUX := PWRFLEX_FEEDBACK_AUX3 / 1.5;
PWRFLEX_FEEDBACK_AUX4 := BUGGY_SPEED_FEEDBACK_OFFSET_AUX * BUGGY_SPEED_FEEDBACK_OFFSET;

// NETWORK 35 (disabled)
// label: //CONVERT ANALOGINPUT1_1 TO AMPS (0-10)

// NETWORK 36
ANA_IN_AUX1 := ANA_INPUT1_1 * 10;
ANA_AMPS := ANA_IN_AUX1 / 32767;

// NETWORK 37 (disabled)
// label: // POWERFLEX AMPS: (1) Vin to INT, (2) INT to Amps (200% DRIVE MAX CURRENT[48A])

// NETWORK 38
ANA_IN_AUX2 := ANA_INPUT1_2 * 10;
PWRFLEX_AMPS_AUX := ANA_IN_AUX2 / 32767;
PWRFLEX_AMPS_AUX := PWRFLEX_AMPS_AUX * 48;
PWRFLEX_AMPS := PWRFLEX_AMPS_AUX / 10;

// NETWORK 39
COGNEX_AUX := In_Sight_Micro_1000_Series;

// NETWORK 40

// NETWORK 41 (disabled)
// label: //-----------------ALARMS-------------------------

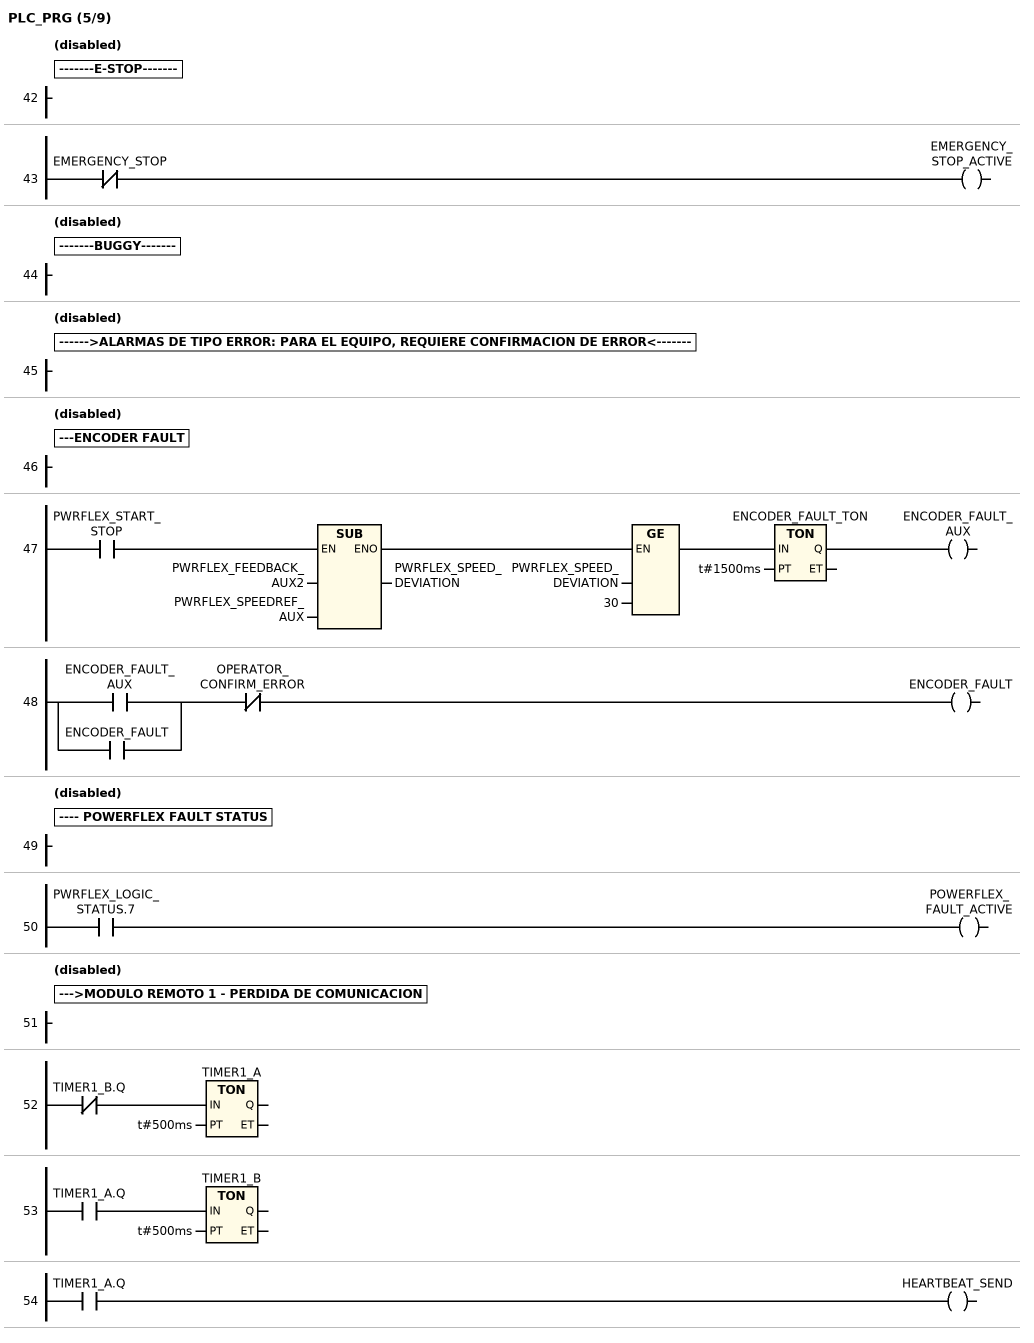
// NETWORK 42 (disabled)
// label: -------E-STOP-------

// NETWORK 43
EMERGENCY_STOP_ACTIVE := NOT EMERGENCY_STOP;

// NETWORK 44 (disabled)
// label: -------BUGGY-------

// NETWORK 45 (disabled)
// label: ------>ALARMAS DE TIPO ERROR: PARA EL EQUIPO, REQUIERE CONFIRMACION DE ERROR<-------

// NETWORK 46 (disabled)
// label: ---ENCODER FAULT

// NETWORK 47
_w3 := PWRFLEX_START_STOP;
IF _w3 THEN PWRFLEX_SPEED_DEVIATION := PWRFLEX_FEEDBACK_AUX2 - PWRFLEX_SPEEDREF_AUX; END_IF
ENCODER_FAULT_TON(IN := _w3 AND PWRFLEX_SPEED_DEVIATION >= 30, PT := t#1500ms); // TON
ENCODER_FAULT_AUX := ENCODER_FAULT_TON.Q;

// NETWORK 48
ENCODER_FAULT := (ENCODER_FAULT_AUX OR ENCODER_FAULT) AND NOT OPERATOR_CONFIRM_ERROR;

// NETWORK 49 (disabled)
// label: ---- POWERFLEX FAULT STATUS

// NETWORK 50
POWERFLEX_FAULT_ACTIVE := PWRFLEX_LOGIC_STATUS.7;

// NETWORK 51 (disabled)
// label: --->MODULO REMOTO 1 - PERDIDA DE COMUNICACION

// NETWORK 52
TIMER1_A(IN := NOT TIMER1_B.Q, PT := t#500ms); // TON

// NETWORK 53
TIMER1_B(IN := TIMER1_A.Q, PT := t#500ms); // TON

// NETWORK 54
HEARTBEAT_SEND := TIMER1_A.Q;

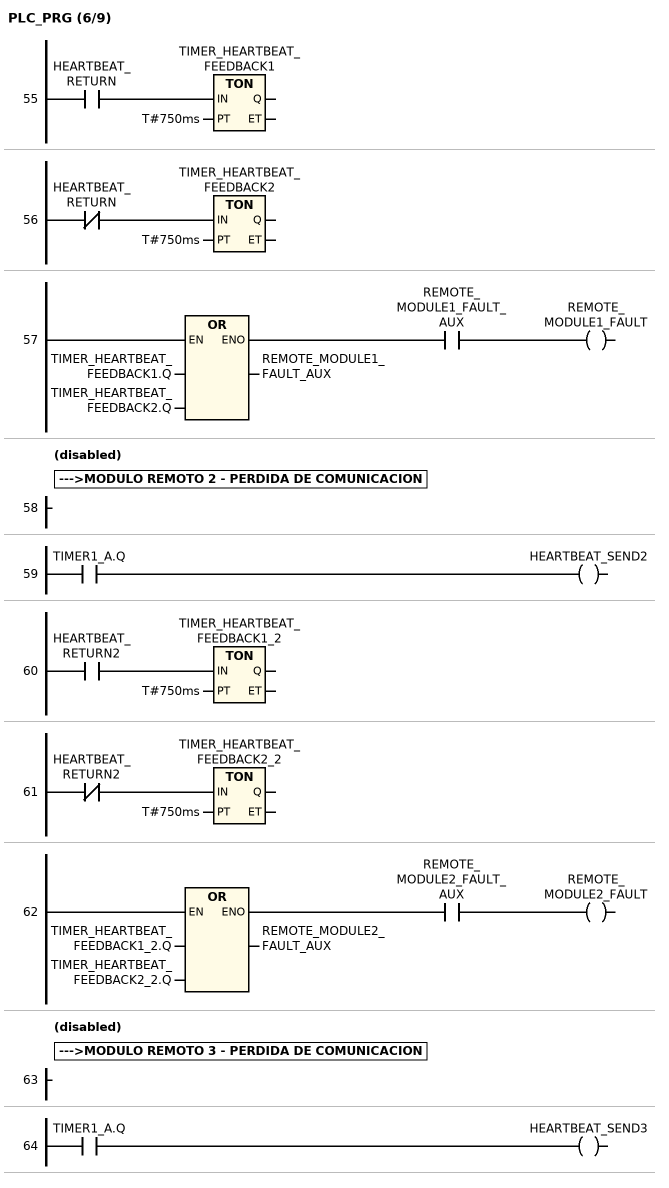
// NETWORK 55
TIMER_HEARTBEAT_FEEDBACK1(IN := HEARTBEAT_RETURN, PT := T#750ms); // TON

// NETWORK 56
TIMER_HEARTBEAT_FEEDBACK2(IN := NOT HEARTBEAT_RETURN, PT := T#750ms); // TON

// NETWORK 57
REMOTE_MODULE1_FAULT_AUX := TIMER_HEARTBEAT_FEEDBACK1.Q OR TIMER_HEARTBEAT_FEEDBACK2.Q;
REMOTE_MODULE1_FAULT := REMOTE_MODULE1_FAULT_AUX;

// NETWORK 58 (disabled)
// label: --->MODULO REMOTO 2 - PERDIDA DE COMUNICACION

// NETWORK 59
HEARTBEAT_SEND2 := TIMER1_A.Q;

// NETWORK 60
TIMER_HEARTBEAT_FEEDBACK1_2(IN := HEARTBEAT_RETURN2, PT := T#750ms); // TON

// NETWORK 61
TIMER_HEARTBEAT_FEEDBACK2_2(IN := NOT HEARTBEAT_RETURN2, PT := T#750ms); // TON

// NETWORK 62
REMOTE_MODULE2_FAULT_AUX := TIMER_HEARTBEAT_FEEDBACK1_2.Q OR TIMER_HEARTBEAT_FEEDBACK2_2.Q;
REMOTE_MODULE2_FAULT := REMOTE_MODULE2_FAULT_AUX;

// NETWORK 63 (disabled)
// label: --->MODULO REMOTO 3 - PERDIDA DE COMUNICACION

// NETWORK 64
HEARTBEAT_SEND3 := TIMER1_A.Q;

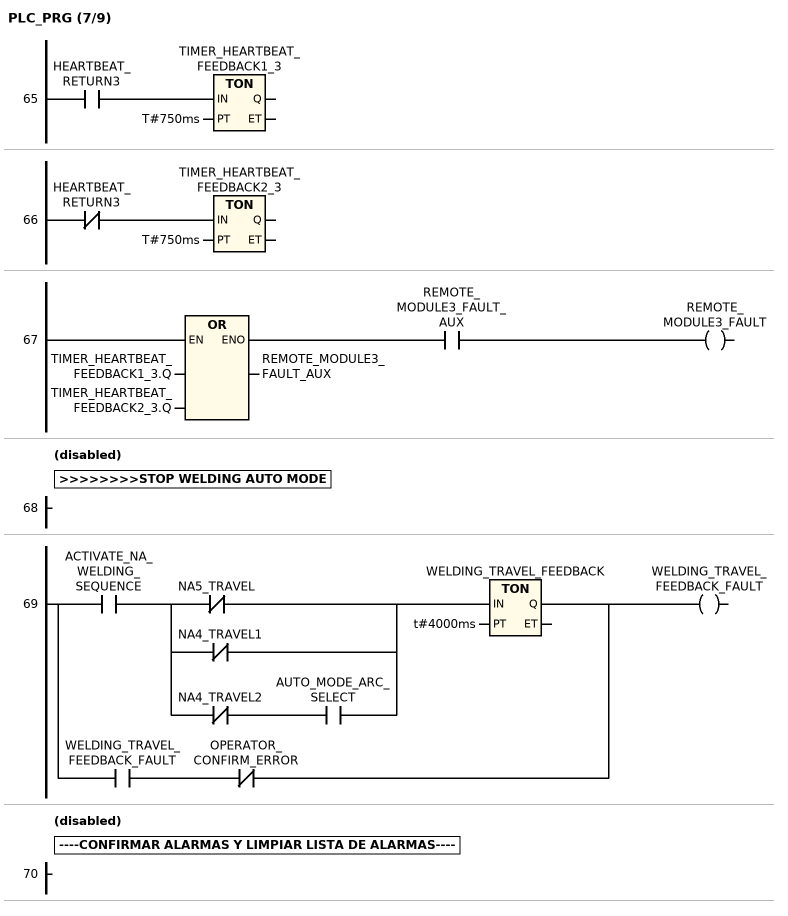
// NETWORK 65
TIMER_HEARTBEAT_FEEDBACK1_3(IN := HEARTBEAT_RETURN3, PT := T#750ms); // TON

// NETWORK 66
TIMER_HEARTBEAT_FEEDBACK2_3(IN := NOT HEARTBEAT_RETURN3, PT := T#750ms); // TON

// NETWORK 67
REMOTE_MODULE3_FAULT_AUX := TIMER_HEARTBEAT_FEEDBACK1_3.Q OR TIMER_HEARTBEAT_FEEDBACK2_3.Q;
REMOTE_MODULE3_FAULT := REMOTE_MODULE3_FAULT_AUX;

// NETWORK 68 (disabled)
// label: >>>>>>>>STOP WELDING AUTO MODE

// NETWORK 69
_w4 := WELDING_TRAVEL_FEEDBACK_FAULT AND NOT OPERATOR_CONFIRM_ERROR;
IF NOT _w4 THEN
    WELDING_TRAVEL_FEEDBACK(IN := ACTIVATE_NA_WELDING_SEQUENCE AND (NOT NA5_TRAVEL OR NOT NA4_TRAVEL1 OR NOT NA4_TRAVEL2 AND AUTO_MODE_ARC_SELECT), PT := t#4000ms); // TON
    _w4 := WELDING_TRAVEL_FEEDBACK.Q;
END_IF
WELDING_TRAVEL_FEEDBACK_FAULT := _w4;

// NETWORK 70 (disabled)
// label: ----CONFIRMAR ALARMAS Y LIMPIAR LISTA DE ALARMAS----

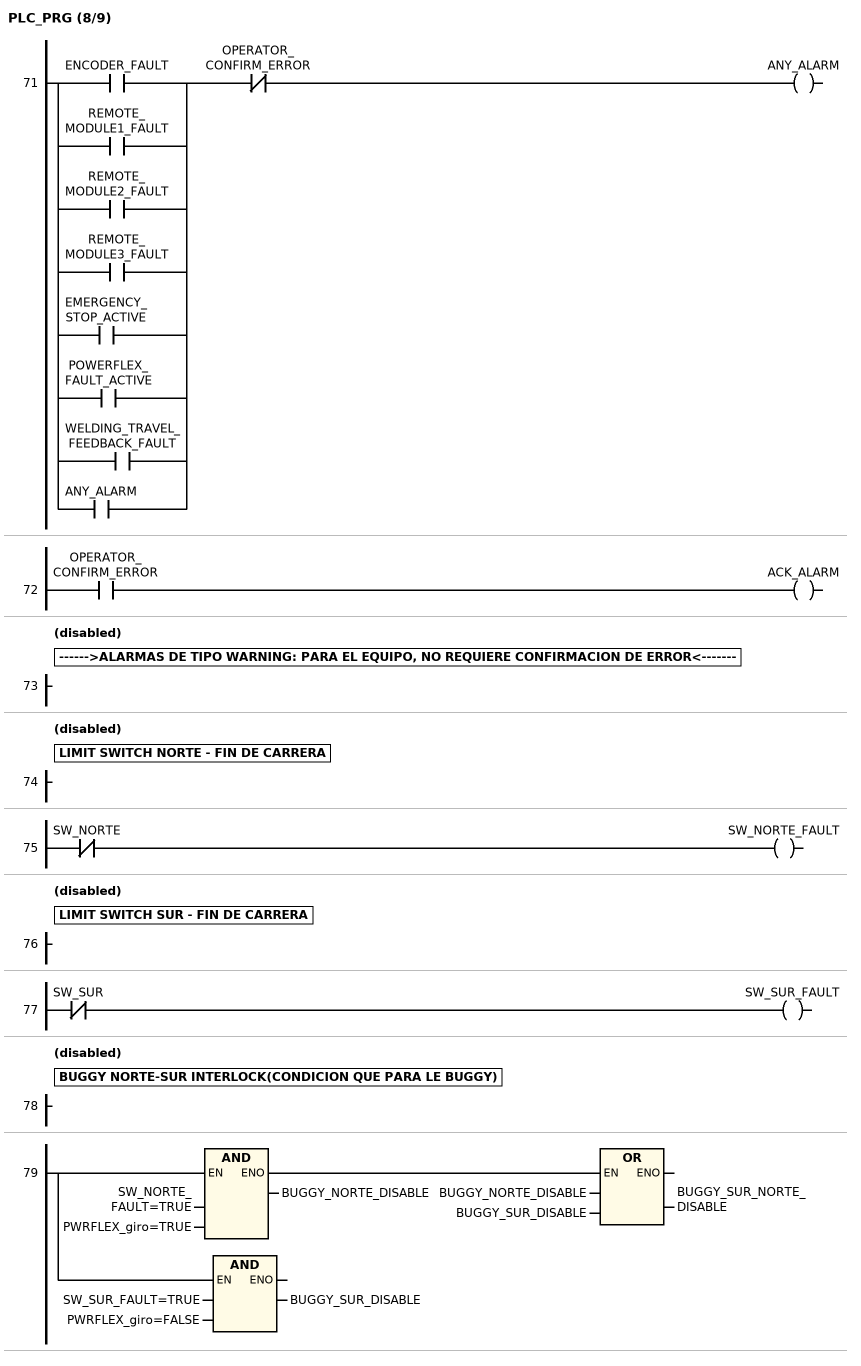
// NETWORK 71
ANY_ALARM := (ENCODER_FAULT OR REMOTE_MODULE1_FAULT OR REMOTE_MODULE2_FAULT OR REMOTE_MODULE3_FAULT OR EMERGENCY_STOP_ACTIVE OR POWERFLEX_FAULT_ACTIVE OR WELDING_TRAVEL_FEEDBACK_FAULT OR ANY_ALARM) AND NOT OPERATOR_CONFIRM_ERROR;

// NETWORK 72
ACK_ALARM := OPERATOR_CONFIRM_ERROR;

// NETWORK 73 (disabled)
// label: ------>ALARMAS DE TIPO WARNING: PARA EL EQUIPO, NO REQUIERE CONFIRMACION DE ERROR<-------

// NETWORK 74 (disabled)
// label: LIMIT SWITCH NORTE - FIN DE CARRERA

// NETWORK 75
SW_NORTE_FAULT := NOT SW_NORTE;

// NETWORK 76 (disabled)
// label: LIMIT SWITCH SUR - FIN DE CARRERA

// NETWORK 77
SW_SUR_FAULT := NOT SW_SUR;

// NETWORK 78 (disabled)
// label: BUGGY NORTE-SUR INTERLOCK(CONDICION QUE PARA LE BUGGY)

// NETWORK 79
BUGGY_NORTE_DISABLE := (SW_NORTE_FAULT=TRUE) AND (PWRFLEX_giro=TRUE);
BUGGY_SUR_NORTE_DISABLE := BUGGY_NORTE_DISABLE OR BUGGY_SUR_DISABLE;
BUGGY_SUR_DISABLE := (SW_SUR_FAULT=TRUE) AND (PWRFLEX_giro=FALSE);

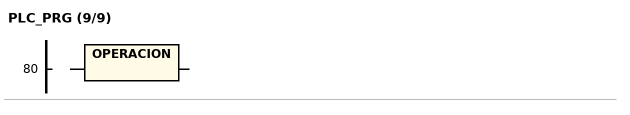
// NETWORK 80
OPERACION();

END_PROGRAM

// Device/Application/OPERACION
PROGRAM OPERACION
VAR
	
//-----------------------------------OPERACION VARS-----------------------------------------//
//-----------TOLVA ON/OFF---------------
//RELAY: L02: C5
HMI_TOLVA_ON: BOOL;
TOLVA_ON: BOOL;

//-----------CAMARA ON/OFF---------------
//RELAY: L02: C6
HMI_CAMARA_ON: BOOL;
CAMARA_ON: BOOL;

//-----------CONTROL ANTORCHA---------------
//HMI
HMI_JOYUP  :BOOL; 
HMI_JOYDOWN  :BOOL; 
HMI_JOY_EJEA :BOOL;
HMI_JOY_EJEB :BOOL;
//JOYSTICK
JOYUP  :BOOL; 
JOYDOWN  :BOOL; 
JOY_EJEA :BOOL;
JOY_EJEB :BOOL;

//LIMIT SWITCHES
SW_ANORTCHA_UP: BOOL;
SW_ANTORCHA_DOWN: BOOL;
SW_ANTORCHA_EJEA: BOOL;
SW_ANTORCHA_EJEB: BOOL;

//CONROL RELAYS (L02: C7-EJEA,C8-EJEB,C9-SUBIR,C10-BAJAR)
ANTORCHA_UP: BOOL;
ANTORCHA_DOWN: BOOL;
ANTORCHA_EJEA: BOOL;
ANTORCHA_EJEB: BOOL;

//--------------ROTADORES------------------
HMI_ROTADORES_EJEA :BOOL;
ROTATORS_EJEA_TOF: TOF;	//OFF DELAY INTERLOCK
HMI_ROTADORES_EJEB :BOOL;
ROTATORS_EJEB_TOF: TOF;	//OFF DELAY INTERLOCK

//INFO
ROTADORES_INFO_MSG :BOOL;

//CONTROL RELAYS
ROTADORES_EJEA_L02_KM3: BOOL;
ROTADORES_EJEB_L02_KM4: BOOL;

//--------------CONVEYORS-------------------
HMI_CONVEYOR_NORTE :BOOL;
CONVEYOR_NORTE_TOF: TOF;	//OFF DELAY INTERLOCK
HMI_CONVEYOR_SUR :BOOL;
CONVEYOR_SUR_TOF: TOF;	//OFF DELAY INTERLOCK

//CONTROL RELAYS
CONVEYOR_NORTE_L02_KM1: BOOL;
CONVEYOR_SUR_L02_KM2: BOOL;

//--------------BOOM-------------------
HMI_BOOM_UP: BOOL;
BOOM_UP_TOF: TOF;	//OFF DELAY INTERLOCK
HMI_BOOM_DOWN: BOOL;
BOOM_DOWN_TOF: TOF;	//OFF DELAY INTERLOCK

//SWITCHES
SW_BOOM_UP: BOOL;
SW_BOOM_DOWN: BOOL;

//CONTROL RELAYS
BOOM_UP_KM5: BOOL;
BOOM_DOWN_KM6: BOOL;

//--------------ASPIRADORA-------------------
HMI_ASPIRADORA: BOOL;
ASPIRADORA_KM7: BOOL;

//---------VALVULAS SISTEMA TIERRAS----------
//RELAYS: L02: C1,C2
//INPUTS:
HMI_VALVULA1: BOOL;
HMI_VALVULA2: BOOL;

//OUTPUTS
RELAY_VALVULA1: BOOL;
RELAY_VALVULA2: BOOL;

//---------MOTOR SISTEMA TIERRAS----------
//RELAYS: L01: RL8-SUBIR, RL9-BAJAR
//INPUTS:
HMI_BRAZO_TIERRAS_UP: BOOL;
BRAZO_TIERRAS_UP_TOF: TOF;	//OFF DELAY INTERLOCK
HMI_BRAZO_TIERRAS_DOWN: BOOL;
BRAZO_TIERRAS_DOWN_TOF: TOF;	//OFF DELAY INTERLOCK

//OUTPUTS
RELAY_BRAZO_TIERRAS_UP: BOOL;
RELAY_BRAZO_TIERRAS_DOWN: BOOL;
END_VAR

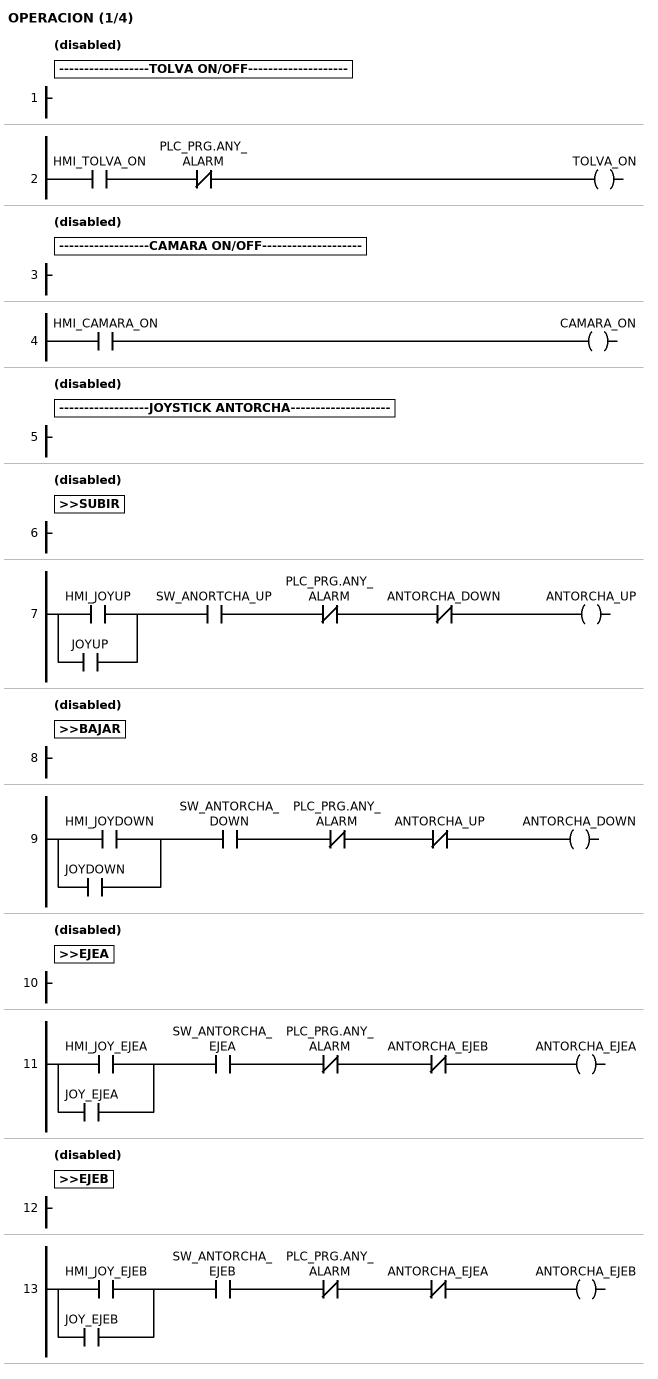
// NETWORK 1 (disabled)
// label: ------------------TOLVA ON/OFF--------------------

// NETWORK 2
TOLVA_ON := HMI_TOLVA_ON AND NOT PLC_PRG.ANY_ALARM;

// NETWORK 3 (disabled)
// label: ------------------CAMARA ON/OFF--------------------

// NETWORK 4
CAMARA_ON := HMI_CAMARA_ON;

// NETWORK 5 (disabled)
// label: ------------------JOYSTICK ANTORCHA--------------------

// NETWORK 6 (disabled)
// label: >>SUBIR

// NETWORK 7
ANTORCHA_UP := (HMI_JOYUP OR JOYUP) AND SW_ANORTCHA_UP AND NOT PLC_PRG.ANY_ALARM AND NOT ANTORCHA_DOWN;

// NETWORK 8 (disabled)
// label: >>BAJAR

// NETWORK 9
ANTORCHA_DOWN := (HMI_JOYDOWN OR JOYDOWN) AND SW_ANTORCHA_DOWN AND NOT PLC_PRG.ANY_ALARM AND NOT ANTORCHA_UP;

// NETWORK 10 (disabled)
// label: >>EJEA

// NETWORK 11
ANTORCHA_EJEA := (HMI_JOY_EJEA OR JOY_EJEA) AND SW_ANTORCHA_EJEA AND NOT PLC_PRG.ANY_ALARM AND NOT ANTORCHA_EJEB;

// NETWORK 12 (disabled)
// label: >>EJEB

// NETWORK 13
ANTORCHA_EJEB := (HMI_JOY_EJEB OR JOY_EJEB) AND SW_ANTORCHA_EJEB AND NOT PLC_PRG.ANY_ALARM AND NOT ANTORCHA_EJEA;

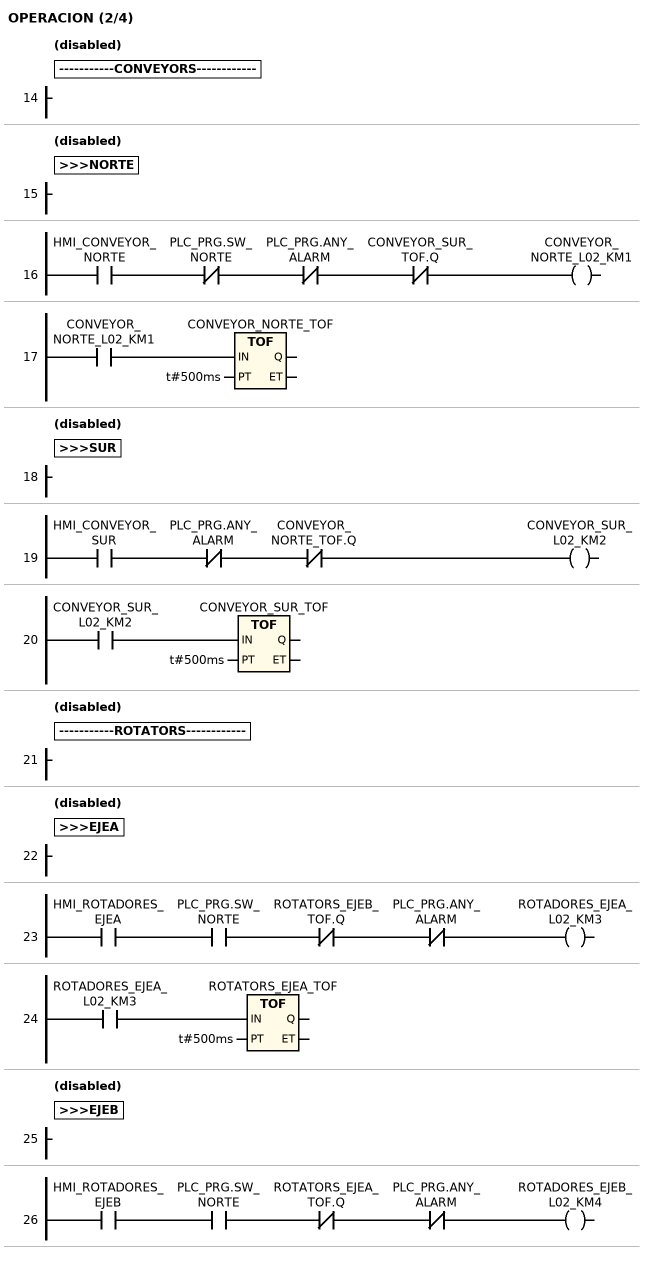
// NETWORK 14 (disabled)
// label: -----------CONVEYORS------------

// NETWORK 15 (disabled)
// label: >>>NORTE

// NETWORK 16
CONVEYOR_NORTE_L02_KM1 := HMI_CONVEYOR_NORTE AND NOT PLC_PRG.SW_NORTE AND NOT PLC_PRG.ANY_ALARM AND NOT CONVEYOR_SUR_TOF.Q;

// NETWORK 17
CONVEYOR_NORTE_TOF(IN := CONVEYOR_NORTE_L02_KM1, PT := t#500ms); // TOF

// NETWORK 18 (disabled)
// label: >>>SUR

// NETWORK 19
CONVEYOR_SUR_L02_KM2 := HMI_CONVEYOR_SUR AND NOT PLC_PRG.ANY_ALARM AND NOT CONVEYOR_NORTE_TOF.Q;

// NETWORK 20
CONVEYOR_SUR_TOF(IN := CONVEYOR_SUR_L02_KM2, PT := t#500ms); // TOF

// NETWORK 21 (disabled)
// label: -----------ROTATORS------------

// NETWORK 22 (disabled)
// label: >>>EJEA

// NETWORK 23
ROTADORES_EJEA_L02_KM3 := HMI_ROTADORES_EJEA AND PLC_PRG.SW_NORTE AND NOT ROTATORS_EJEB_TOF.Q AND NOT PLC_PRG.ANY_ALARM;

// NETWORK 24
ROTATORS_EJEA_TOF(IN := ROTADORES_EJEA_L02_KM3, PT := t#500ms); // TOF

// NETWORK 25 (disabled)
// label: >>>EJEB

// NETWORK 26
ROTADORES_EJEB_L02_KM4 := HMI_ROTADORES_EJEB AND PLC_PRG.SW_NORTE AND NOT ROTATORS_EJEA_TOF.Q AND NOT PLC_PRG.ANY_ALARM;

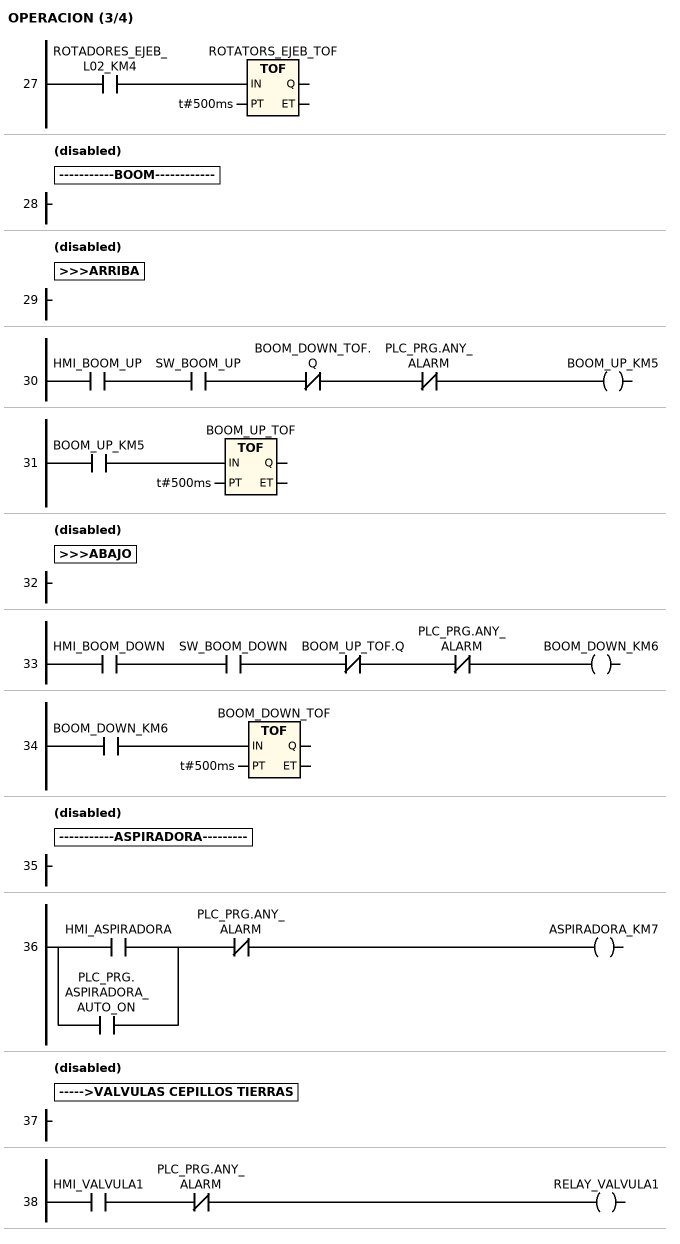
// NETWORK 27
ROTATORS_EJEB_TOF(IN := ROTADORES_EJEB_L02_KM4, PT := t#500ms); // TOF

// NETWORK 28 (disabled)
// label: -----------BOOM------------

// NETWORK 29 (disabled)
// label: >>>ARRIBA

// NETWORK 30
BOOM_UP_KM5 := HMI_BOOM_UP AND SW_BOOM_UP AND NOT BOOM_DOWN_TOF.Q AND NOT PLC_PRG.ANY_ALARM;

// NETWORK 31
BOOM_UP_TOF(IN := BOOM_UP_KM5, PT := t#500ms); // TOF

// NETWORK 32 (disabled)
// label: >>>ABAJO

// NETWORK 33
BOOM_DOWN_KM6 := HMI_BOOM_DOWN AND SW_BOOM_DOWN AND NOT BOOM_UP_TOF.Q AND NOT PLC_PRG.ANY_ALARM;

// NETWORK 34
BOOM_DOWN_TOF(IN := BOOM_DOWN_KM6, PT := t#500ms); // TOF

// NETWORK 35 (disabled)
// label: -----------ASPIRADORA---------

// NETWORK 36
ASPIRADORA_KM7 := (HMI_ASPIRADORA OR PLC_PRG.ASPIRADORA_AUTO_ON) AND NOT PLC_PRG.ANY_ALARM;

// NETWORK 37 (disabled)
// label: ----->VALVULAS CEPILLOS TIERRAS

// NETWORK 38
RELAY_VALVULA1 := HMI_VALVULA1 AND NOT PLC_PRG.ANY_ALARM;

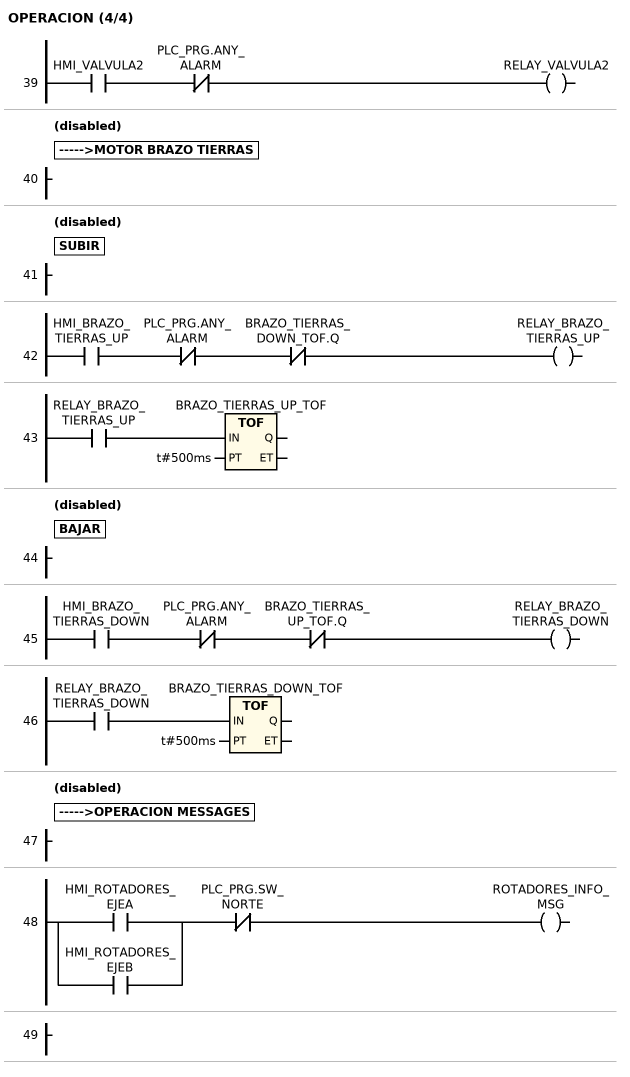
// NETWORK 39
RELAY_VALVULA2 := HMI_VALVULA2 AND NOT PLC_PRG.ANY_ALARM;

// NETWORK 40 (disabled)
// label: ----->MOTOR BRAZO TIERRAS

// NETWORK 41 (disabled)
// label: SUBIR

// NETWORK 42
RELAY_BRAZO_TIERRAS_UP := HMI_BRAZO_TIERRAS_UP AND NOT PLC_PRG.ANY_ALARM AND NOT BRAZO_TIERRAS_DOWN_TOF.Q;

// NETWORK 43
BRAZO_TIERRAS_UP_TOF(IN := RELAY_BRAZO_TIERRAS_UP, PT := t#500ms); // TOF

// NETWORK 44 (disabled)
// label: BAJAR

// NETWORK 45
RELAY_BRAZO_TIERRAS_DOWN := HMI_BRAZO_TIERRAS_DOWN AND NOT PLC_PRG.ANY_ALARM AND NOT BRAZO_TIERRAS_UP_TOF.Q;

// NETWORK 46
BRAZO_TIERRAS_DOWN_TOF(IN := RELAY_BRAZO_TIERRAS_DOWN, PT := t#500ms); // TOF

// NETWORK 47 (disabled)
// label: ----->OPERACION MESSAGES

// NETWORK 48
ROTADORES_INFO_MSG := (HMI_ROTADORES_EJEA OR HMI_ROTADORES_EJEB) AND NOT PLC_PRG.SW_NORTE;

// NETWORK 49

END_PROGRAM

// Device/Application/CSVMON_FILE_GEN
PROGRAM CSVMON_FILE_GEN
VAR
(* 
======>instalar librerias:
1)network(OSCAT 1.2.1.0)
2)CAA FILE 3.5.7.0
*)	
//STATES	
STATE: USINT:=0;	//0=IDLE,1=CREATE FILE,2=GENERATE HEADER,3=DAQ,4=FTP SEND FILE

//FILE GEN
START_MON: BOOL;


//FILE NAME
fileDIR: FILENAME:='./Param_MON/';
//fileNAME: FILENAME;  //-ORIGINAL
fileNAME: FILENAME:='C0'; //-TEST
fileEXTENSION: FILENAME:='.csv';
fileBUFFER: FILENAME;
fileFULL: FILENAME;

//FILE HEADER
//DATOS_TUBO: STRING;  -ORIGINAL
DATOS_TUBO: STRING:='ID12345'; //-TEST


COLUMN_ID_CTU: CTU;
COLUMN_ID: WORD;
COLUMN_ID_AUX: WORD;
COLUMN_ID_RESET: BOOL;

MONITOR_ROW_BUFFER: STRING;
DATA1: REAL;
DATA2: REAL;
DATACONV_BUFFER: STRING;
ROW_STRING_READY: BOOL:=FALSE;

TXT_LINE_END: WORD;
TXT_LINE_END_AUX: STRING;


//FILE VARS
fileOPEN_START : BOOL;
fileOPEN_ENABLE :BOOL;
openFILE_FTRIG : F_TRIG;

	sFileName 		: FILE.CAA.FILENAME;
	sFileNameCopy 	: FILE.CAA.FILENAME;	
	FileOpen 		: File.Open;
	FileClose		: File.Close;
	FileCopy		: File.Copy;
	GetFileSize		: File.GetSize;
	GetFileTime		: File.GetTime;
	FileRead		: File.Read;
	FileWrite		: File.Write;
	SetFilePos		: File.SetPos;
	GetFilePos		: File.GetPos;	

	hfile			: FILE.CAA.HANDLE;
	sWriteLine		: STRING(128);
	sReadLine		: STRING;	
	dtModification 	: DATE_AND_TIME;
	udiFileSize		: __XWORD;
	xError			: BOOL := FALSE;
	xInit			: BOOL := FALSE;
	xTestDone		: BOOL := FALSE;
	xStartTest		: BOOL := FALSE; (* true, if a button is pressed *)

	FILE_CREATE_ENABLE: BOOL;
	FILE_CREATE_ST_CTRL: USINT:=0;
	FILE_CREATE_DONE: BOOL:=FALSE;
	FILE_CREATE_BUSY: BOOL:=FALSE;
	FILE_CREATE_ERROR: BOOL:=FALSE;
	
	HEADER_BUFFER: STRING;
	WRITE_HEADER_DONE: BOOL:=FALSE;
	WRITE_HEADER_ERROR: BOOL:=FALSE;
	HEADER_ST_CTRL: USINT:=0;
	
	SAMPLING_CLOCK: TON;
	
	
	DAQ_ST_CTRL: USINT;
	DAQ_WRITE_DONE: BOOL;
	DAQ_WRITE_ERROR: BOOL;
	DAQ_WRITE_STATE_DONE: BOOL;
	DAQ_WRITE_GOTO_NEXT_STATE: BOOL;
	
//SYSTEM TIME	
actualTime: SysTime64;
ActualTimeEx: SystemTimeDate;
RdCurTimeEx: CurTimeEx;



//----------------------------FTP VARS------------------------------//
FTP_CLIENT0: OSCAT_NETWORK.FTP_CLIENT;
//FTP_RISING_TRIG0: R_TRIG;
FTP_FALLING_TRIG0: F_TRIG;
//IN
FTP_ENABLE: BOOL;
FTP_START: BOOL:=0;

FTP_CTRL: BOOL:=0; //0=UPLOAD, 1=DOWNLOAD
FTP_ACTIVE: BOOL:=0; //PASSIVE = 0 (recommended)/ ACTIVE = 1)
FTP_FILE_DELETE: BOOL:=1; //0=KEEP , 1=DELETE
FTP_TIMEOUT: TIME:=T#30000MS; //30seg


//OUT
FTP_DONE: BOOL;
FTP_BUSY: BOOL;
FTP_ERROR_C: DWORD;
FTP_ERROR_T: BYTE;




//MISC
ALWAYS_OFF: BOOL:=FALSE;
TEST_BIT: BOOL:=FALSE;

END_VAR
VAR // added by the converter: edge detectors and wires of the graphical bodies
    _w1, _w2, _w3, _w4, _w5, _w6, _w7 : BOOL;
END_VAR

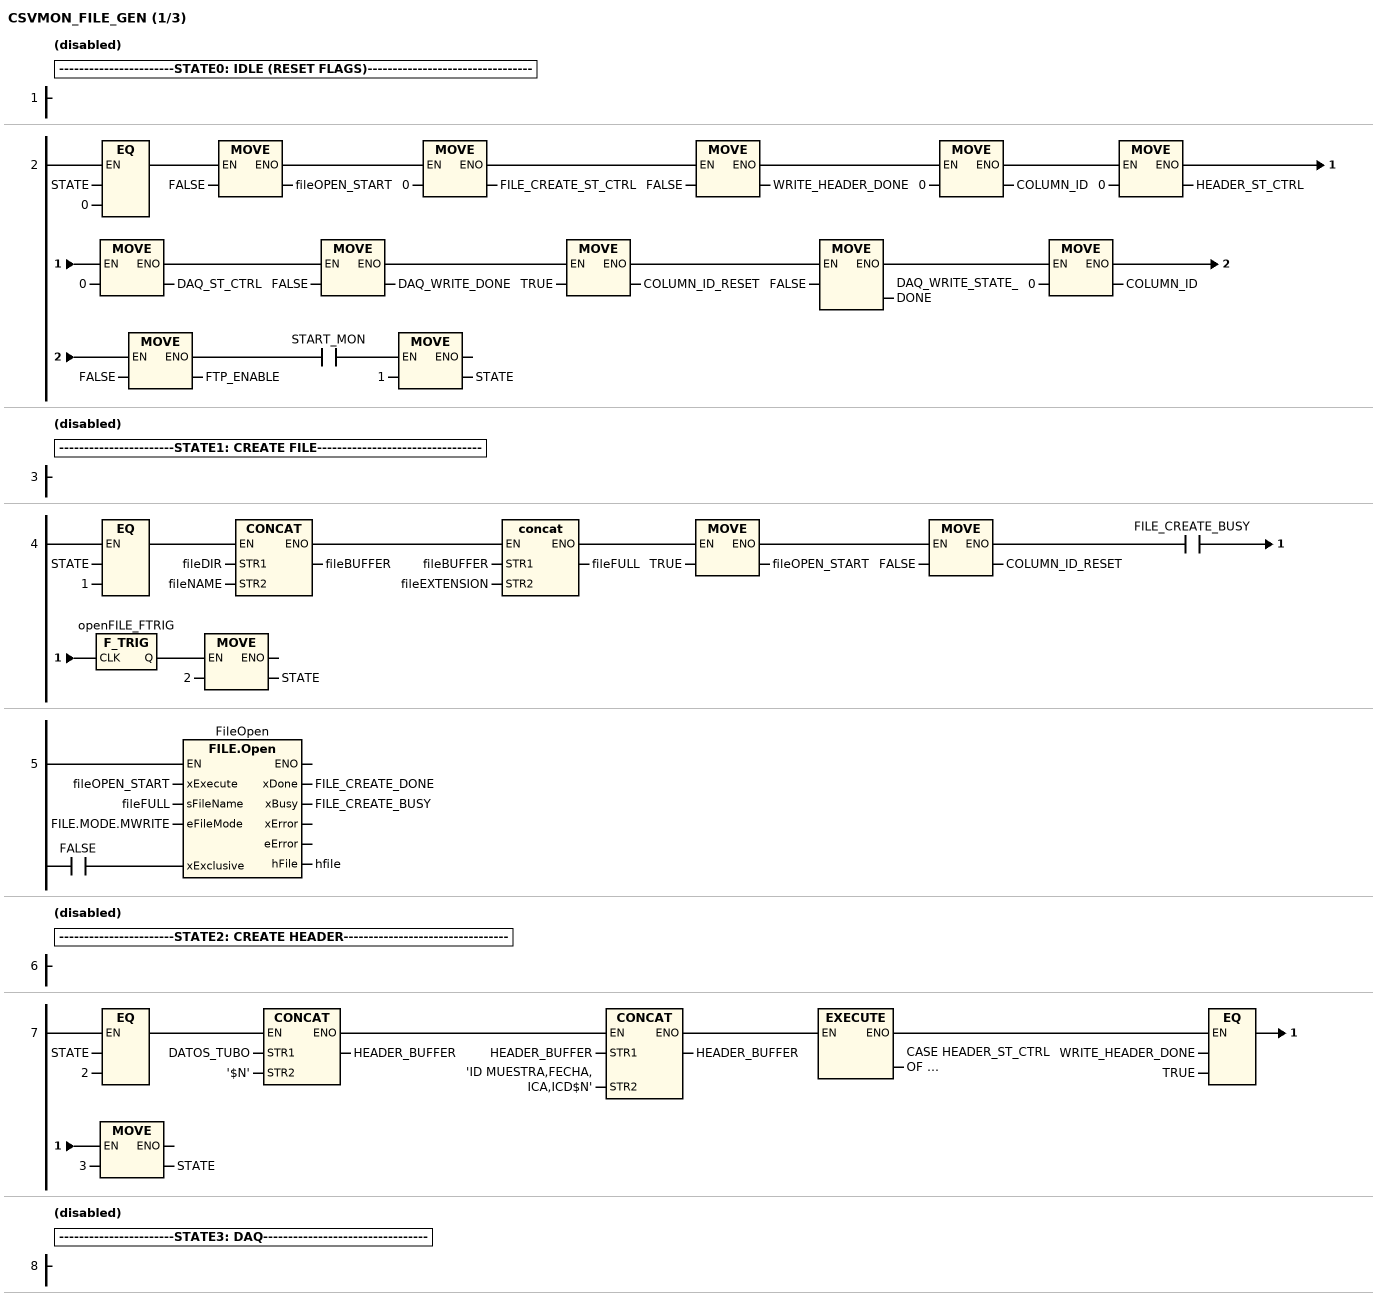
// NETWORK 1 (disabled)
// label: -----------------------STATE0: IDLE (RESET FLAGS)---------------------------------

// NETWORK 2
_w1 := STATE = 0;
IF _w1 THEN fileOPEN_START := FALSE; END_IF
IF _w1 THEN FILE_CREATE_ST_CTRL := 0; END_IF
IF _w1 THEN WRITE_HEADER_DONE := FALSE; END_IF
IF _w1 THEN COLUMN_ID := 0; END_IF
IF _w1 THEN HEADER_ST_CTRL := 0; END_IF
IF _w1 THEN DAQ_ST_CTRL := 0; END_IF
IF _w1 THEN DAQ_WRITE_DONE := FALSE; END_IF
IF _w1 THEN COLUMN_ID_RESET := TRUE; END_IF
IF _w1 THEN DAQ_WRITE_STATE_DONE := FALSE; END_IF
IF _w1 THEN COLUMN_ID := 0; END_IF
IF _w1 THEN FTP_ENABLE := FALSE; END_IF
IF _w1 AND START_MON THEN STATE := 1; END_IF

// NETWORK 3 (disabled)
// label: -----------------------STATE1: CREATE FILE---------------------------------

// NETWORK 4
_w2 := STATE = 1;
IF _w2 THEN fileBUFFER := CONCAT(STR1 := fileDIR, STR2 := fileNAME); END_IF
IF _w2 THEN fileFULL := concat(STR1 := fileBUFFER, STR2 := fileEXTENSION); END_IF
IF _w2 THEN fileOPEN_START := TRUE; END_IF
IF _w2 THEN COLUMN_ID_RESET := FALSE; END_IF
openFILE_FTRIG(CLK := _w2 AND FILE_CREATE_BUSY); // F_TRIG
IF openFILE_FTRIG.Q THEN STATE := 2; END_IF

// NETWORK 5
FileOpen(
    xExecute := fileOPEN_START,
    sFileName := fileFULL,
    eFileMode := FILE.MODE.MWRITE,
    xExclusive := FALSE,
    xDone => FILE_CREATE_DONE,
    xBusy => FILE_CREATE_BUSY,
    hFile => hfile); // FILE.Open

// NETWORK 6 (disabled)
// label: -----------------------STATE2: CREATE HEADER---------------------------------

// NETWORK 7
_w3 := STATE = 2;
IF _w3 THEN HEADER_BUFFER := CONCAT(STR1 := DATOS_TUBO, STR2 := '$N'); END_IF
IF _w3 THEN HEADER_BUFFER := CONCAT(STR1 := HEADER_BUFFER, STR2 := 'ID MUESTRA,FECHA,ICA,ICD$N'); END_IF
IF _w3 THEN
    
    CASE HEADER_ST_CTRL OF
    	0:
    		   sWriteLine := HEADER_BUFFER;
    		   FileWrite(xExecute:= TRUE,hFile:= hfile, pBuffer:= ADR(sWriteLine), szSize:= INT_TO_UDINT(LEN(sWriteLine)));
    		   IF FileWrite.xDone = TRUE THEN
    		 	//  HEADER_ST_CTRL := 1; //ORIGINAL
    			   HEADER_ST_CTRL := 2;
    			   FileWrite(xExecute:= FALSE);
    		   ELSIF FileOpen.xError = TRUE THEN
    			  WRITE_HEADER_ERROR:= TRUE;
    			   FileWrite(xExecute:= FALSE);
    		   END_IF
    	1:	   
    		      FileClose(xExecute:= TRUE, hFile:= hfile);
    	   IF FileClose.xDone = TRUE THEN
    		   
    		   HEADER_ST_CTRL := 2;
    		   FileClose(xExecute:= FALSE);
    	   ELSIF FileClose.xError = TRUE THEN
    		   WRITE_HEADER_ERROR:= TRUE;
    		   FileClose(xExecute:= FALSE);
    	   END_IF
    	2:
    		WRITE_HEADER_DONE :=TRUE;
    END_CASE
END_IF
IF _w3 AND WRITE_HEADER_DONE = TRUE THEN STATE := 3; END_IF

// NETWORK 8 (disabled)
// label: -----------------------STATE3: DAQ---------------------------------

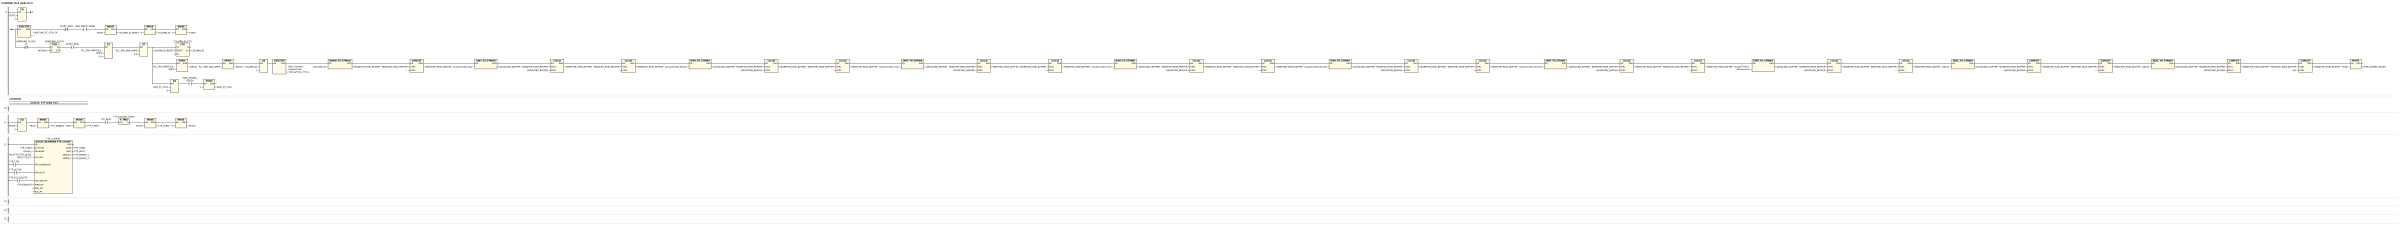
// NETWORK 9
_w4 := STATE = 3;
IF _w4 THEN
    CASE DAQ_ST_CTRL OF
    	0: //IDLE
    	IF START_MON=FALSE THEN	   
    		
    		DAQ_ST_CTRL := 3;
    	END_IF
    	
    	1: // Append a string to the file.
    	   ROW_STRING_READY:=FALSE;
    	   sWriteLine := MONITOR_ROW_BUFFER;
    	   FileWrite(xExecute:= TRUE, hFile:= hfile, pBuffer:=ADR(sWriteLine), szSize:= INT_TO_UDINT(LEN(sWriteLine)));
    	   IF FileWrite.xDone = TRUE THEN
    DAQ_ST_CTRL := 4;
    		   FileWrite(xExecute:= FALSE);
    	   ELSIF FileWrite.xError = TRUE THEN
    		   DAQ_ST_CTRL:= 6;
    		   FileWrite(xExecute:= FALSE);
    	   END_IF
    	   
    	3: // Close the file.
    	   FileClose(xExecute:= TRUE, hFile:= hfile);
    	   IF FileClose.xDone = TRUE THEN
    		   DAQ_ST_CTRL := 4;
    		   FileClose(xExecute:= FALSE);
    		   DAQ_WRITE_DONE:= TRUE;
    		      
    	   ELSIF FileClose.xError = TRUE THEN
    		   DAQ_ST_CTRL:= 7;
    		   FileClose(xExecute:= FALSE);
    	   END_IF
    	  
        4://DONE
    	
    	   DAQ_ST_CTRL:= 0;
    END_CASE
END_IF
IF _w4 AND NOT START_MON AND DAQ_WRITE_DONE THEN COLUMN_ID_RESET := TRUE; END_IF
IF _w4 AND NOT START_MON AND DAQ_WRITE_DONE THEN COLUMN_ID := 0; END_IF
IF _w4 AND NOT START_MON AND DAQ_WRITE_DONE THEN STATE := 4; END_IF
SAMPLING_CLOCK(IN := _w4 AND NOT SAMPLING_CLOCK.Q, PT := t#250ms); // TON
_w5 := SAMPLING_CLOCK.Q AND START_MON AND PLC_PRG.PWRFLEX_AMPS > 0.0 AND PLC_PRG.ANA_AMPS > 0.2;
COLUMN_ID_CTU(CU := _w5, RESET := COLUMN_ID_RESET, CV => COLUMN_ID); // CTU
IF _w5 THEN DATA1 := PLC_PRG.PWRFLEX_AMPS; END_IF
IF _w5 THEN DATA2 := PLC_PRG.ANA_AMPS; END_IF
IF _w5 AND COLUMN_ID >= 1 THEN RdCurTimeEx(SystemTime:=ActualTime, TimeDate:=ActualTimeEx); END_IF
IF _w5 AND COLUMN_ID >= 1 THEN MONITOR_ROW_BUFFER := WORD_TO_STRING(COLUMN_ID); END_IF
IF _w5 AND COLUMN_ID >= 1 THEN MONITOR_ROW_BUFFER := CONCAT(STR1 := MONITOR_ROW_BUFFER, STR2 := ','); END_IF
IF _w5 AND COLUMN_ID >= 1 THEN DATACONV_BUFFER := UINT_TO_STRING(ActualTimeEx.Day); END_IF
IF _w5 AND COLUMN_ID >= 1 THEN
    MONITOR_ROW_BUFFER := concat(STR1 := MONITOR_ROW_BUFFER, STR2 := DATACONV_BUFFER);
END_IF
IF _w5 AND COLUMN_ID >= 1 THEN MONITOR_ROW_BUFFER := concat(STR1 := MONITOR_ROW_BUFFER, STR2 := '.'); END_IF
IF _w5 AND COLUMN_ID >= 1 THEN DATACONV_BUFFER := UINT_TO_STRING(ActualTimeEx.Month); END_IF
IF _w5 AND COLUMN_ID >= 1 THEN
    MONITOR_ROW_BUFFER := concat(STR1 := MONITOR_ROW_BUFFER, STR2 := DATACONV_BUFFER);
END_IF
IF _w5 AND COLUMN_ID >= 1 THEN MONITOR_ROW_BUFFER := concat(STR1 := MONITOR_ROW_BUFFER, STR2 := '.'); END_IF
IF _w5 AND COLUMN_ID >= 1 THEN DATACONV_BUFFER := UINT_TO_STRING(ActualTimeEx.Year); END_IF
IF _w5 AND COLUMN_ID >= 1 THEN
    MONITOR_ROW_BUFFER := concat(STR1 := MONITOR_ROW_BUFFER, STR2 := DATACONV_BUFFER);
END_IF
IF _w5 AND COLUMN_ID >= 1 THEN MONITOR_ROW_BUFFER := concat(STR1 := MONITOR_ROW_BUFFER, STR2 := ' '); END_IF
IF _w5 AND COLUMN_ID >= 1 THEN DATACONV_BUFFER := UINT_TO_STRING(ActualTimeEx.Hour); END_IF
IF _w5 AND COLUMN_ID >= 1 THEN
    MONITOR_ROW_BUFFER := concat(STR1 := MONITOR_ROW_BUFFER, STR2 := DATACONV_BUFFER);
END_IF
IF _w5 AND COLUMN_ID >= 1 THEN MONITOR_ROW_BUFFER := concat(STR1 := MONITOR_ROW_BUFFER, STR2 := ':'); END_IF
IF _w5 AND COLUMN_ID >= 1 THEN DATACONV_BUFFER := UINT_TO_STRING(ActualTimeEx.Minute); END_IF
IF _w5 AND COLUMN_ID >= 1 THEN
    MONITOR_ROW_BUFFER := concat(STR1 := MONITOR_ROW_BUFFER, STR2 := DATACONV_BUFFER);
END_IF
IF _w5 AND COLUMN_ID >= 1 THEN MONITOR_ROW_BUFFER := concat(STR1 := MONITOR_ROW_BUFFER, STR2 := ':'); END_IF
IF _w5 AND COLUMN_ID >= 1 THEN DATACONV_BUFFER := UINT_TO_STRING(ActualTimeEx.Second); END_IF
IF _w5 AND COLUMN_ID >= 1 THEN
    MONITOR_ROW_BUFFER := concat(STR1 := MONITOR_ROW_BUFFER, STR2 := DATACONV_BUFFER);
END_IF
IF _w5 AND COLUMN_ID >= 1 THEN MONITOR_ROW_BUFFER := concat(STR1 := MONITOR_ROW_BUFFER, STR2 := '.'); END_IF
IF _w5 AND COLUMN_ID >= 1 THEN DATACONV_BUFFER := UINT_TO_STRING(ActualTimeEx.Milliseconds); END_IF
IF _w5 AND COLUMN_ID >= 1 THEN
    MONITOR_ROW_BUFFER := concat(STR1 := MONITOR_ROW_BUFFER, STR2 := DATACONV_BUFFER);
END_IF
IF _w5 AND COLUMN_ID >= 1 THEN MONITOR_ROW_BUFFER := concat(STR1 := MONITOR_ROW_BUFFER, STR2 := ','); END_IF
IF _w5 AND COLUMN_ID >= 1 THEN DATACONV_BUFFER := REAL_TO_STRING(DATA1); END_IF
IF _w5 AND COLUMN_ID >= 1 THEN
    MONITOR_ROW_BUFFER := CONCAT(STR1 := MONITOR_ROW_BUFFER, STR2 := DATACONV_BUFFER);
END_IF
IF _w5 AND COLUMN_ID >= 1 THEN MONITOR_ROW_BUFFER := CONCAT(STR1 := MONITOR_ROW_BUFFER, STR2 := ','); END_IF
IF _w5 AND COLUMN_ID >= 1 THEN DATACONV_BUFFER := REAL_TO_STRING(DATA2); END_IF
IF _w5 AND COLUMN_ID >= 1 THEN
    MONITOR_ROW_BUFFER := CONCAT(STR1 := MONITOR_ROW_BUFFER, STR2 := DATACONV_BUFFER);
END_IF
IF _w5 AND COLUMN_ID >= 1 THEN MONITOR_ROW_BUFFER := CONCAT(STR1 := MONITOR_ROW_BUFFER, STR2 := '$N'); END_IF
IF _w5 AND COLUMN_ID >= 1 THEN ROW_STRING_READY := TRUE; END_IF
IF (_w5 AND DAQ_ST_CTRL = 0) AND ROW_STRING_READY THEN DAQ_ST_CTRL := 1; END_IF

// NETWORK 10 (disabled)
// label: -----------------------STATE4: FTP SEND FILE---------------------------------

// NETWORK 11
_w6 := STATE = 4;
IF _w6 THEN FTP_ENABLE := TRUE; END_IF
IF _w6 THEN FTP_START := TRUE; END_IF
FTP_FALLING_TRIG0(CLK := _w6 AND FTP_BUSY); // F_TRIG
_w7 := FTP_FALLING_TRIG0.Q;
IF _w7 THEN FTP_START := FALSE; END_IF
IF _w7 THEN STATE := 0; END_IF

// NETWORK 12
FTP_CLIENT0(
    ACTIVATE := FTP_START,
    FILENAME := fileFULL,
    FTP_URL := 'ftp://FTP_TEST:@192.168.5.211:21/',
    FTP_DOWNLOAD := FTP_CTRL,
    FTP_ACTIV := FTP_ACTIVE,
    FILE_DELETE := FTP_FILE_DELETE,
    TIMEOUT := FTP_TIMEOUT,
    DONE => FTP_DONE,
    BUSY => FTP_BUSY,
    ERROR_C => FTP_ERROR_C,
    ERROR_T => FTP_ERROR_T); // OSCAT_NETWORK.FTP_CLIENT

// NETWORK 13

// NETWORK 14

// NETWORK 15

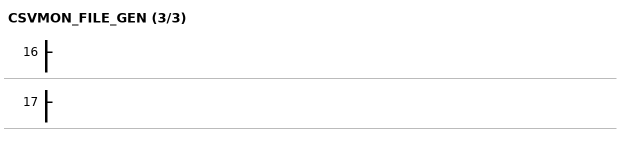
// NETWORK 16

// NETWORK 17

END_PROGRAM

// Device/Application/PRINCIPAL
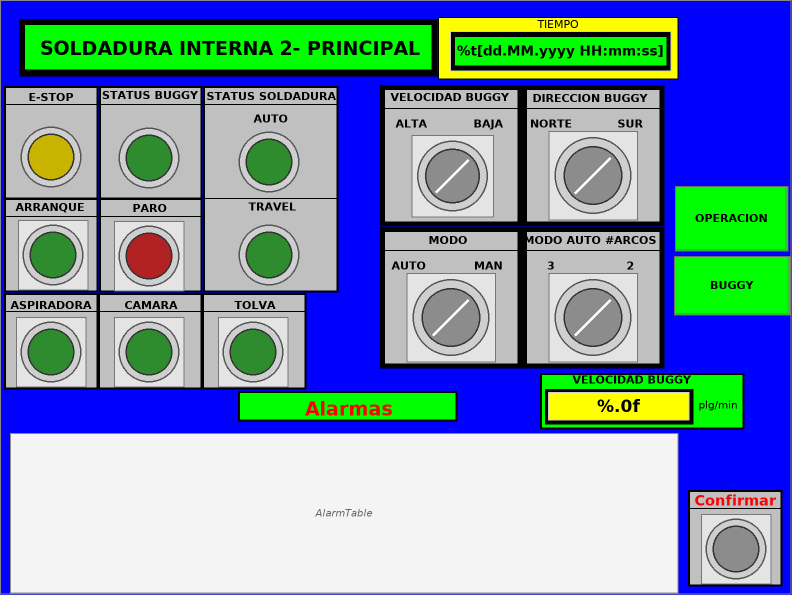
VISUALIZATION PRINCIPAL  // 792x595
    Rectangle (203,86 135x206)
    Rectangle (99,86 103x113)
    Rectangle (688,490 94x96)
    Rectangle (4,86 94x113)
    Lamp1 (16,122 70x70), variable: PLC_PRG.ANY_ALARM, style: Lamp-Lamp1-Yellow
    Lamp1 (114,123 70x70), variable: PLC_PRG.PWRFLEX_START_STOP, style: Lamp-Lamp1-Green
    Label (1,84 100x27), "E-STOP"
    Label (100,82 100x27), "STATUS BUGGY"
    Line (98,104) (337,104)
    Rectangle (540,373 204x56)
    Rectangle (545,389 148x35)
    Label (557,365 150x30), "VELOCIDAD BUGGY"
    Group (19,19 411x57)
        Group (0,0 418x57)
            Rectangle (0,0 418x57)
            Rectangle (5,5 408x46)
        Label (79,10 260x39), "SOLDADORA INTERNA 1"
    Group (19,19 418x57)
        Rectangle (0,0 418x57)
        Rectangle (5,5 408x46)
    Rectangle (19,19 418x57)
    Rectangle (24,24 408x46)
    Label (32,29 396x39), "SOLDADURA INTERNA 2- PRINCIPAL"
    Rectangle (438,17 240x62)
    Label (508,11 100x27), "TIEMPO"
    Textfield (450,31 221x40)
    Rectangle (454,36 213x30), "%t[dd.MM.yyyy HH:mm:ss]"
    Line (5,104) (99,104)
    Textfield (697,390 42x30), "plg/min"
    Textfield (548,392 141x28), "%.0f", text variable: PLC_PRG.PWRFLEX_FEEDBACK_AUX4
    Rectangle (380,85 142x141)
    Line (381,108) (520,108)
    Rectangle (392,115 39x18), "ALTA"
    Rectangle (469,115 39x18), "BAJA"
    RotarySwitch (408,135 89x82), variable: PLC_PRG.BUGGY_SPEED_SELECTOR, behaviour: TOGGLE, style: Switch-RotarySwitch-Gray
    Label (375,84 150x27), "VELOCIDAD BUGGY"
    Group (238,391 219x33)
        Rectangle (0,0 219x30)
        Label (7,3 208x30), "Alarmas"
    AlarmTable (10,433 668x160)
        p1521930926: __All
        p1663851261: __All
        p2607059081: PLC_PRG.ACK_ALARM
    Rectangle (522,85 142x141)
    Line (523,108) (663,108)
    Rectangle (529,115 44x18), "NORTE"
    Rectangle (611,115 39x18), "SUR"
    Label (515,85 150x27), "DIRECCION BUGGY"
    RotarySwitch (548,131 90x89), variable: PLC_PRG.PWRFLEX_giro, behaviour: TOGGLE, style: Switch-RotarySwitch-Gray
    PushSwitch (701,514 70x70), variable: PLC_PRG.OPERATOR_CONFIRM_ERROR, behaviour: TAP, style: Switch-PushSwitch-Gray
    Label (690,478 91x45), "Confirmar"
    Line (688,508) (782,508)
    Rectangle (4,293 94x96)
    Label (1,292 100x27), "ASPIRADORA"
    Line (4,311) (98,311)
    PushSwitch (16,317 70x70), variable: OPERACION.HMI_ASPIRADORA, behaviour: TOGGLE, style: Switch-PushSwitch-Green
    Button (675,186 113x65), "OPERACION"
        OnMouseDown:  Assign=OPERACION, Type=Assignment
    Button (674,256 116x59), "BUGGY"
        OnMouseDown:  Assign=BUGGY, Type=Assignment
    Rectangle (380,227 142x141)
    Line (381,250) (521,250)
    Rectangle (387,257 44x18), "AUTO"
    Rectangle (469,257 39x18), "MAN"
    Label (373,227 150x27), "MODO"
    RotarySwitch (406,273 90x89), variable: PLC_PRG.HMI_AUTO_MODE, behaviour: TOGGLE, style: Switch-RotarySwitch-Gray
    Label (207,83 129x27), "STATUS SOLDADURA"
    Line (203,88) (203,183)
    Lamp1 (234,127 70x70), variable: PLC_PRG.AUTO_MODE_PERMISSIVES_OK, style: Lamp-Lamp1-Green
    Lamp1 (234,220 70x70), variable: PLC_PRG.ALL_NA_TRAVEL_OK, style: Lamp-Lamp1-Green
    Rectangle (252,110 38x18), "AUTO"
    Rectangle (244,198 57x18), "TRAVEL"
    Line (204,198) (336,198)
    Rectangle (99,198 103x94)
    Rectangle (4,198 94x94)
    PushSwitch (18,220 70x70), variable: PLC_PRG.PWRFLEX_OPERATOR_START, behaviour: TAP, style: Switch-PushSwitch-Green
    PushSwitch (114,221 70x70), variable: PLC_PRG.HMI_PWRFLEX_OPERATOR_STOP, behaviour: TAP, style: Switch-PushSwitch-Red
    Label (0,194 100x27), "ARRANQUE"
    Label (100,195 100x27), "PARO"
    Line (5,216) (203,216)
    Rectangle (98,293 104x96)
    Label (101,292 100x27), "CAMARA"
    Line (98,311) (202,311)
    PushSwitch (114,317 70x70), variable: OPERACION.HMI_CAMARA_ON, behaviour: TOGGLE, style: Switch-PushSwitch-Green
    Rectangle (202,293 104x96)
    Label (205,292 100x27), "TOLVA"
    Line (202,311) (306,311)
    PushSwitch (218,317 70x70), variable: OPERACION.HMI_TOLVA_ON, behaviour: TOGGLE, style: Switch-PushSwitch-Green
    Rectangle (522,227 142x141)
    Line (523,250) (663,250)
    Rectangle (529,257 44x18), "3"
    Rectangle (611,257 39x18), "2"
    Label (515,227 150x27), "MODO AUTO #ARCOS"
    RotarySwitch (548,273 90x89), variable: PLC_PRG.AUTO_MODE_ARC_SELECT, behaviour: TOGGLE, style: Switch-RotarySwitch-Gray
END_VISUALIZATION

// Device/Application/Analog_Test
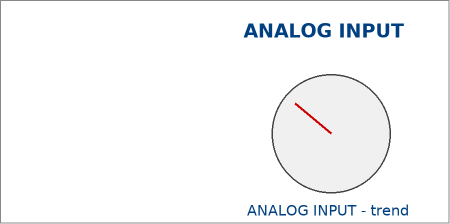
VISUALIZATION Analog_Test  // 450x224
    Meter180 (214,74 234x119), value: PLC_PRG.ANA_AMPS, style: Meter-Meter180-Green, scale format: %.1f, scale 0..10
    Label (222,16 204x30), "ANALOG INPUT"
    Label (219,199 218x23), "ANALOG INPUT - trend"
END_VISUALIZATION

// Device/Application/Drive_Test
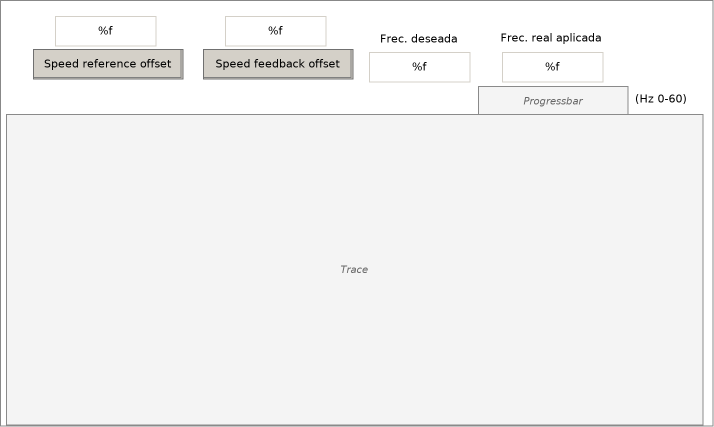
VISUALIZATION Drive_Test  // 714x427
    Progressbar (478,86 150x30), variable: PLC_PRG.PWRFLEX_FEEDBACK
    Trace (6,114 697x311)
    Textfield (369,52 101x30), "%f", text variable: PLC_PRG.PWRFLEX_SPEEDREF_AUX
    Label (368,24 102x30), "Frec. deseada"
    Textfield (502,52 101x30), "%f", text variable: PLC_PRG.PWRFLEX_FEEDBACK_AUX2
    Label (500,23 102x30), "Frec. real aplicada"
    Label (610,84 102x30), "(Hz 0-60)"
    Button (203,49 150x30), "Speed feedback offset"
        OnMouseClick: write PLC_PRG.BUGGY_SPEED_FEEDBACK_OFFSET via VisuDialogs.NumpadExtended
    Textfield (225,16 101x30), "%f", text variable: PLC_PRG.BUGGY_SPEED_FEEDBACK_OFFSET
    Button (33,49 150x30), "Speed reference offset"
        OnMouseClick: write PLC_PRG.BUGGY_SPEED_REFERENCE_OFFSET via VisuDialogs.NumpadExtended
    Textfield (55,16 101x30), "%f", text variable: PLC_PRG.BUGGY_SPEED_REFERENCE_OFFSET
END_VISUALIZATION

// Device/Application/Test_DAQ
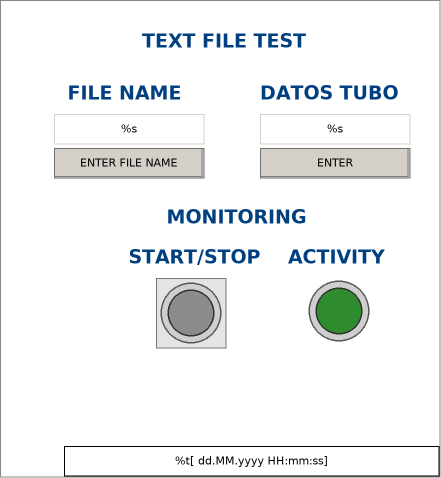
VISUALIZATION Test_DAQ  // 441x478
    Label (89,26 270x30), "TEXT FILE TEST"
    Rectangle (64,446 375x30), "%t[ dd.MM.yyyy HH:mm:ss]"
    Button (54,148 150x30), "ENTER FILE NAME"
        OnMouseClick: write CSVMON_FILE_GEN.fileNAME via VisuDialogs.Keypad
    Textfield (54,114 150x30), "%s", text variable: CSVMON_FILE_GEN.fileNAME
    Label (57,78 135x30), "FILE NAME"
    Label (262,78 135x30), "DATOS TUBO"
    Textfield (260,114 150x30), "%s", text variable: CSVMON_FILE_GEN.DATOS_TUBO
    Button (260,148 150x30), "ENTER"
        OnMouseDown: write CSVMON_FILE_GEN.DATOS_TUBO via VisuDialogs.Keypad
    Lamp1 (304,276 70x70), variable: CSVMON_FILE_GEN.START_MON, style: Lamp-Lamp1-Green
    Label (169,202 135x30), "MONITORING"
    Label (269,242 135x30), "ACTIVITY"
    PushSwitch (156,278 70x70), variable: CSVMON_FILE_GEN.START_MON, behaviour: TOGGLE, style: Switch-PushSwitch-Gray
    Label (127,242 135x30), "START/STOP"
END_VISUALIZATION

// Device/Application/OPERACION
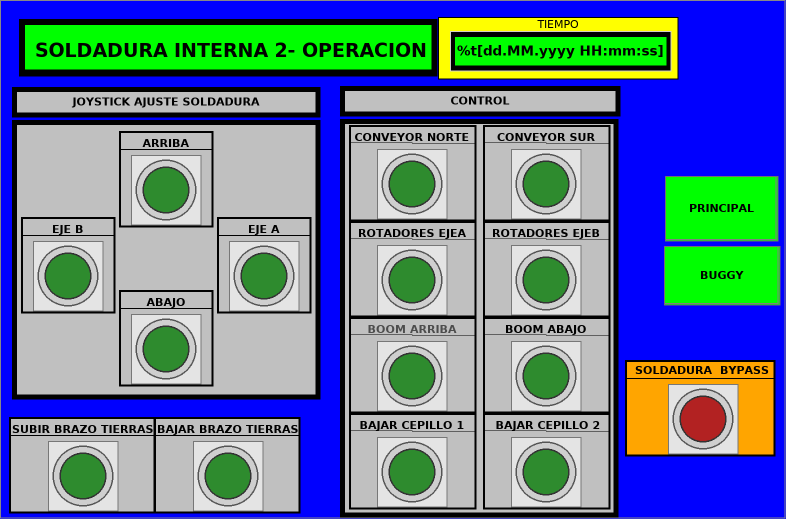
VISUALIZATION OPERACION  // 786x519
    Group (19,11 659x68)
        Group (0,8 411x57)
            Group (0,0 418x57)
                Rectangle (0,0 418x57)
                Rectangle (5,5 408x46)
            Label (79,10 260x39), "SOLDADORA INTERNA 1"
        Rectangle (419,6 240x62)
        Label (489,0 100x27), "TIEMPO"
        Textfield (431,20 221x40)
        Rectangle (435,25 213x30), "%t[dd.MM.yyyy HH:mm:ss]"
    Group (19,19 411x57)
        Group (0,0 418x57)
            Rectangle (0,0 418x57)
            Rectangle (5,5 408x46)
        Label (79,10 260x39), "SOLDADORA INTERNA 1"
    Group (19,19 418x57)
        Rectangle (0,0 418x57)
        Rectangle (5,5 408x46)
    Rectangle (19,19 418x57)
    Rectangle (24,24 408x46)
    Rectangle (438,17 240x62)
    Label (508,11 100x27), "TIEMPO"
    Textfield (450,31 221x40)
    Rectangle (454,36 213x30), "%t[dd.MM.yyyy HH:mm:ss]"
    Rectangle (12,120 308x279)
    Rectangle (119,131 94x96)
    Label (116,130 100x27), "ARRIBA"
    Line (119,149) (213,149)
    PushSwitch (131,155 70x70), variable: OPERACION.HMI_JOYUP, behaviour: TAP, style: Switch-PushSwitch-Green
    Rectangle (119,290 94x96)
    Label (116,289 100x27), "ABAJO"
    Line (119,308) (213,308)
    PushSwitch (131,314 70x70), variable: OPERACION.HMI_JOYDOWN, behaviour: TAP, style: Switch-PushSwitch-Green
    Rectangle (21,217 94x96)
    Label (18,216 100x27), "EJE B"
    Line (21,235) (115,235)
    PushSwitch (33,241 70x70), variable: OPERACION.HMI_JOY_EJEB, behaviour: TAP, style: Switch-PushSwitch-Green
    Rectangle (217,217 94x96)
    Label (214,216 100x27), "EJE A"
    Line (217,235) (311,235)
    PushSwitch (229,241 70x70), variable: OPERACION.HMI_JOY_EJEA, behaviour: TAP, style: Switch-PushSwitch-Green
    Rectangle (12,87 308x30), "JOYSTICK AJUSTE SOLDADURA"
    Rectangle (340,119 278x398)
    Rectangle (349,125 127x96)
    Label (354,124 116x27), "CONVEYOR NORTE"
    Line (349,142) (475,143)
    PushSwitch (377,149 70x70), variable: OPERACION.HMI_CONVEYOR_NORTE, behaviour: TAP, style: Switch-PushSwitch-Green
    Rectangle (483,125 127x96)
    Label (488,124 116x27), "CONVEYOR SUR"
    Line (483,142) (609,143)
    PushSwitch (511,149 70x70), variable: OPERACION.HMI_CONVEYOR_SUR, behaviour: TAP, style: Switch-PushSwitch-Green
    Rectangle (349,221 127x96)
    Label (354,220 116x27), "ROTADORES EJEA"
    Line (349,238) (475,239)
    PushSwitch (377,245 70x70), variable: OPERACION.HMI_ROTADORES_EJEA, behaviour: TAP, style: Switch-PushSwitch-Green
    Rectangle (483,221 127x96)
    Label (488,220 116x27), "ROTADORES EJEB"
    Line (483,238) (609,239)
    PushSwitch (511,245 70x70), variable: OPERACION.HMI_ROTADORES_EJEB, behaviour: TAP, style: Switch-PushSwitch-Green
    Rectangle (340,86 280x30), "CONTROL"
    Rectangle (349,317 127x96)
    Label (354,316 116x27), "BOOM ARRIBA"
    Line (349,334) (475,335)
    PushSwitch (377,341 70x70), variable: OPERACION.HMI_BOOM_UP, behaviour: TAP, style: Switch-PushSwitch-Green
    Rectangle (483,317 127x96)
    Label (488,316 116x27), "BOOM ABAJO"
    Line (483,334) (609,335)
    PushSwitch (511,341 70x70), variable: OPERACION.HMI_BOOM_DOWN, behaviour: TAP, style: Switch-PushSwitch-Green
    Label (33,31 396x39), "SOLDADURA INTERNA 2- OPERACION"
    Button (665,176 113x65), "PRINCIPAL"
        OnMouseDown:  Assign=PRINCIPAL, Type=Assignment
    Button (664,246 116x59), "BUGGY"
        OnMouseDown:  Assign=BUGGY, Type=Assignment
    Rectangle (349,413 127x96)
    Label (354,412 116x27), "BAJAR CEPILLO 1"
    Line (349,430) (475,431)
    PushSwitch (377,437 70x70), variable: OPERACION.HMI_VALVULA1, behaviour: TOGGLE, style: Switch-PushSwitch-Green
    Rectangle (483,413 127x96)
    Label (488,412 116x27), "BAJAR CEPILLO 2"
    Line (483,430) (609,431)
    PushSwitch (511,437 70x70), variable: OPERACION.HMI_VALVULA2, behaviour: TOGGLE, style: Switch-PushSwitch-Green
    Rectangle (9,417 146x96)
    Label (8,416 150x27), "SUBIR BRAZO TIERRAS"
    Line (10,435) (155,435)
    PushSwitch (48,441 70x70), variable: OPERACION.HMI_BRAZO_TIERRAS_UP, behaviour: TAP, style: Switch-PushSwitch-Green
    Rectangle (154,417 146x96)
    Label (153,416 150x27), "BAJAR BRAZO TIERRAS"
    Line (155,435) (300,435)
    PushSwitch (193,441 70x70), variable: OPERACION.HMI_BRAZO_TIERRAS_DOWN, behaviour: TAP, style: Switch-PushSwitch-Green
    Rectangle (625,360 150x96)
    Label (620,357 164x27), "SOLDADURA BYPASS"
    Line (625,378) (774,378)
    PushSwitch (668,384 70x70), variable: PLC_PRG.AUTO_MODE_BYPASS, behaviour: TOGGLE, style: Switch-PushSwitch-Red
END_VISUALIZATION

// Device/Application/BUGGY
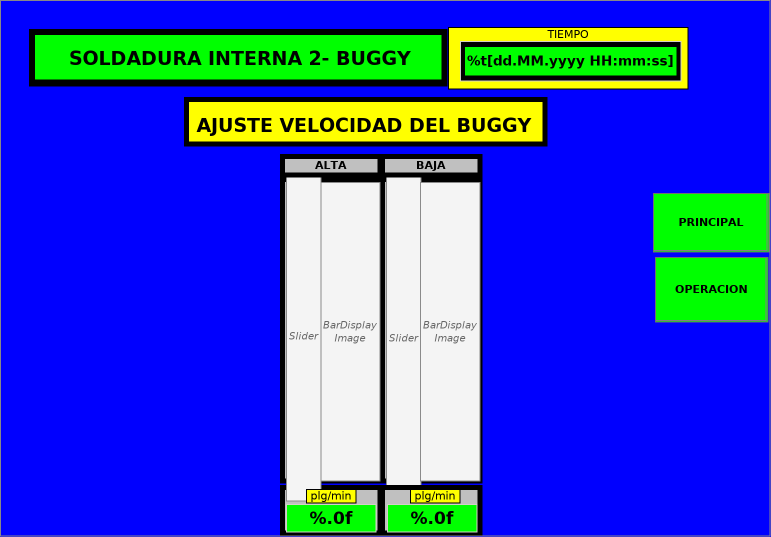
VISUALIZATION BUGGY  // 771x537
    Rectangle (184,97 363x49)
    Group (29,29 411x57)
        Group (0,0 418x57)
            Rectangle (0,0 418x57)
            Rectangle (5,5 408x46)
        Label (79,10 260x39), "SOLDADORA INTERNA 1"
    Group (29,29 418x57)
        Rectangle (0,0 418x57)
        Rectangle (5,5 408x46)
    Rectangle (29,29 418x57)
    Rectangle (34,34 408x46)
    Label (42,39 396x39), "SOLDADURA INTERNA 2- BUGGY"
    Rectangle (448,27 240x62)
    Label (518,21 100x27), "TIEMPO"
    Textfield (460,41 221x40)
    Rectangle (464,46 213x30), "%t[dd.MM.yyyy HH:mm:ss]"
    Line (262,182)
    Line (262,322)
    Rectangle (380,177 102x306)
    Line (362,182)
    Slider (386,173 35x330), variable: PLC_PRG.BUGGY_SPEED_SLOW, scale 15..50
    BarDisplayImage (420,182 60x299), value: PLC_PRG.BUGGY_SPEED_SLOW, style: BarDisplayImage-Yellow, scale format: %i, scale 15..50
    Rectangle (380,485 102x50)
    Textfield (387,504 90x28), "%.0f", text variable: PLC_PRG.BUGGY_SPEED_SLOW
    Rectangle (380,154 102x23), "BAJA"
    Rectangle (280,485 102x50)
    Rectangle (280,177 102x306)
    BarDisplayImage (320,182 60x299), value: PLC_PRG.BUGGY_SPEED_FAST, style: BarDisplayImage-Yellow, scale format: %i, scale 50..500
    Slider (286,171 35x330), variable: PLC_PRG.BUGGY_SPEED_FAST, scale 50..500
    Rectangle (280,154 102x23), "ALTA"
    Textfield (286,504 90x28), "%.0f", text variable: PLC_PRG.BUGGY_SPEED_FAST
    Textfield (306,489 50x14), "plg/min"
    Textfield (410,489 50x14), "plg/min"
    Button (655,257 113x65), "OPERACION"
        OnMouseDown:  Assign=OPERACION, Type=Assignment
    Button (653,193 116x59), "PRINCIPAL"
        OnMouseDown:  Assign=PRINCIPAL, Type=Assignment
    Label (176,102 376x47), "AJUSTE VELOCIDAD DEL BUGGY"
END_VISUALIZATION

(* text list System (id | default)
  Apr | Apr
  April | April
  Aug | Aug
  August | August
  Dec | Dec
  December | December
  Feb | Feb
  February | February
  Fri | Fri
  Friday | Friday
  Jan | Jan
  January | January
  Jul | Jul
  July | July
  Jun | Jun
  June | June
  Mar | Mar
  March | March
  May | May
  May_3Letter | May
  Mon | Mon
  Monday | Monday
  Nov | Nov
  November | November
  Oct | Oct
  October | October
  Sat | Sat
  Saturday | Saturday
  Sep | Sep
  September | September
  Sun | Sun
  Sunday | Sunday
  Thu | Thu
  Thursday | Thursday
  Tue | Tue
  Tuesday | Tuesday
  Wed | Wed
  Wednesday | Wednesday
   |  *)

(* text list AlarmGroup (id | default)
  20 | L2: ERROR COMUNICACION MODULO GABINETE AUXILIAR,ANTORCHAS
  19 | INFO MODO AUTO: BUGGY DIRECCION NORTE, VELOCIDAD LENTA
  18 | ERROR EN GENERACION DE ARCO
  17 | LIMITE BOOM INFERIOR ALCANZADO
  16 | LIMITE BOOM SUPERIOR ALCANZADO
  15 | LIMITE CABEZAL ANTORCHA EJEB ALCANZADO
  14 | LIMITE CABEZAL ANTORCHA EJEA ALCANZADO
  13 | LIMITE CABEZAL ANTORCHA INFERIOR ALCANZADO
  12 | LIMITE CABEZAL ANTORCHA SUPERIOR ALCANZADO
  11 | PARA ACCIONAR ROTADORES, MUEVA EL BUGGY HACIA EL SUR
  10 | L1: ERROR COMUNICACION MODULO GABINETE VARIADOR & FUERZA
  9 | FALLA DRIVE MOTOR BUGGY 
  8 | PRESIONE EL BOTON CONFIRMAR PARA RESTABLECER
  7 | PARO DE EMERGENCIA EXTERNO ACTIVO
  6 | L0: ERROR COMUNICACION MODULO DETRAS HMI PRINCIPAL
  5 | BUGGY LIMITE DE CARRERA SUR ALCANZADO
  4 | BUGGY LIMTE DE CARRERA NORTE ALCANZADO
  3 | ERROR DE SINCRONIZACION BUGGY:REVISAR ENCODER
  2 | NOTIFICACION DE MENSAGE
  1 | NOTIFICACION DE ALERTA1
  0 | NOTIFICACION DE ERROR1
   |  *)
